                                        [[-9.42606,952.141,714.465],[0.876922,0.168711,0.443186,0.0782947],[-1,1,-1,1],[5409.45,9E+09,9E+09,9E+09,9E+09,9E+09]],
                                        [[-9.41231,953.154,714.855],[0.877775,0.167301,0.442197,0.0773528],[-1,1,-1,1],[5407.45,9E+09,9E+09,9E+09,9E+09,9E+09]],
                                        [[-9.39801,954.16,715.244],[0.878624,0.16588,0.441207,0.0764259],[-1,1,-1,1],[5405.45,9E+09,9E+09,9E+09,9E+09,9E+09]],
                                        [[-9.38345,955.166,715.628],[0.879465,0.16447,0.440214,0.0755183],[-1,1,-1,1],[5403.45,9E+09,9E+09,9E+09,9E+09,9E+09]],
                                        [[-9.3692,956.176,716.011],[0.8803,0.163055,0.43922,0.0746309],[-1,1,-1,1],[5401.45,9E+09,9E+09,9E+09,9E+09,9E+09]],
                                        [[-9.35551,957.184,716.389],[0.881131,0.161641,0.438224,0.0737555],[-1,1,-1,1],[5399.45,9E+09,9E+09,9E+09,9E+09,9E+09]],
                                        [[-9.34535,958.198,716.761],[0.881958,0.160216,0.437227,0.0728897],[-1,1,-1,1],[5397.45,9E+09,9E+09,9E+09,9E+09,9E+09]],
                                        [[-9.33447,959.205,717.131],[0.882781,0.158787,0.436228,0.0720344],[-1,1,-1,1],[5395.45,9E+09,9E+09,9E+09,9E+09,9E+09]],
                                        [[-9.32008,960.217,717.498],[0.883599,0.157353,0.435228,0.0711963],[-1,1,-1,1],[5393.45,9E+09,9E+09,9E+09,9E+09,9E+09]],
                                        [[-9.30747,961.231,717.863],[0.884416,0.155903,0.434226,0.070355],[-1,1,-1,1],[5391.45,9E+09,9E+09,9E+09,9E+09,9E+09]],
                                        [[-9.29394,962.246,718.223],[0.885229,0.154452,0.433221,0.0695209],[-1,1,-1,1],[5389.45,9E+09,9E+09,9E+09,9E+09,9E+09]],
                                        [[-9.27922,963.255,718.579],[0.88604,0.152992,0.432214,0.0686898],[-1,1,-1,1],[5387.45,9E+09,9E+09,9E+09,9E+09,9E+09]],
                                        [[-9.26511,964.273,718.932],[0.886848,0.151509,0.431207,0.0678638],[-1,1,-1,1],[5385.45,9E+09,9E+09,9E+09,9E+09,9E+09]],
                                        [[-9.25676,965.291,719.283],[0.887657,0.15,0.4302,0.0670376],[-1,1,-1,1],[5383.45,9E+09,9E+09,9E+09,9E+09,9E+09]],
                                        [[-9.24412,966.308,719.631],[0.888456,0.148507,0.429189,0.0662374],[-1,1,-1,1],[5381.45,9E+09,9E+09,9E+09,9E+09,9E+09]],
                                        [[-9.23401,967.325,719.976],[0.889257,0.146977,0.428179,0.0654321],[-1,1,-1,1],[5379.45,9E+09,9E+09,9E+09,9E+09,9E+09]],
                                        [[-9.22588,968.345,720.318],[0.890054,0.145446,0.427167,0.064639],[-1,1,-1,1],[5377.45,9E+09,9E+09,9E+09,9E+09,9E+09]],
                                        [[-9.21433,969.364,720.656],[0.890847,0.143908,0.426152,0.0638457],[-1,1,-1,1],[5375.45,9E+09,9E+09,9E+09,9E+09,9E+09]],
                                        [[-9.20663,970.383,720.989],[0.891638,0.142368,0.425133,0.0630512],[-1,1,-1,1],[5373.45,9E+09,9E+09,9E+09,9E+09,9E+09]],
                                        [[-9.19797,971.403,721.317],[0.892429,0.140797,0.424113,0.0622536],[-1,1,-1,1],[5371.45,9E+09,9E+09,9E+09,9E+09,9E+09]],
                                        [[-9.18923,972.429,721.644],[0.893216,0.139218,0.423091,0.061457],[-1,1,-1,1],[5369.45,9E+09,9E+09,9E+09,9E+09,9E+09]],
                                        [[-9.18339,973.457,721.968],[0.894004,0.13761,0.422068,0.0606508],[-1,1,-1,1],[5367.45,9E+09,9E+09,9E+09,9E+09,9E+09]],
                                        [[-9.1751,974.477,722.287],[0.894787,0.13601,0.42104,0.0598502],[-1,1,-1,1],[5365.45,9E+09,9E+09,9E+09,9E+09,9E+09]],
                                        [[-9.1676,975.509,722.603],[0.895569,0.134397,0.420009,0.0590409],[-1,1,-1,1],[5363.45,9E+09,9E+09,9E+09,9E+09,9E+09]],
                                        [[-9.15948,976.535,722.914],[0.896348,0.132767,0.418977,0.0582357],[-1,1,-1,1],[5361.45,9E+09,9E+09,9E+09,9E+09,9E+09]],
                                        [[-9.15505,977.568,723.219],[0.897127,0.131111,0.417943,0.0574251],[-1,1,-1,1],[5359.45,9E+09,9E+09,9E+09,9E+09,9E+09]],
                                        [[-9.1446,978.598,723.524],[0.897904,0.129432,0.416907,0.056606],[-1,1,-1,1],[5357.45,9E+09,9E+09,9E+09,9E+09,9E+09]],
                                        [[-9.1363,979.625,723.822],[0.898678,0.127747,0.415867,0.0557895],[-1,1,-1,1],[5355.45,9E+09,9E+09,9E+09,9E+09,9E+09]],
                                        [[-9.1268,980.66,724.115],[0.899451,0.126043,0.414825,0.0549606],[-1,1,-1,1],[5353.45,9E+09,9E+09,9E+09,9E+09,9E+09]],
                                        [[-9.12389,981.693,724.406],[0.900221,0.12434,0.413778,0.0541259],[-1,1,-1,1],[5351.45,9E+09,9E+09,9E+09,9E+09,9E+09]],
                                        [[-9.12032,982.72,724.689],[0.900987,0.12262,0.41273,0.0532925],[-1,1,-1,1],[5349.45,9E+09,9E+09,9E+09,9E+09,9E+09]],
                                        [[-9.11677,983.752,724.97],[0.90175,0.120895,0.411678,0.0524628],[-1,1,-1,1],[5347.45,9E+09,9E+09,9E+09,9E+09,9E+09]],
                                        [[-9.11474,984.782,725.248],[0.902507,0.119183,0.410621,0.0516391],[-1,1,-1,1],[5345.45,9E+09,9E+09,9E+09,9E+09,9E+09]],
                                        [[-9.11064,985.807,725.519],[0.903261,0.11746,0.409561,0.0508105],[-1,1,-1,1],[5343.45,9E+09,9E+09,9E+09,9E+09,9E+09]],
                                        [[-9.10221,986.836,725.788],[0.90401,0.115747,0.408497,0.0499893],[-1,1,-1,1],[5341.45,9E+09,9E+09,9E+09,9E+09,9E+09]],
                                        [[-9.09653,987.866,726.051],[0.904755,0.114033,0.407429,0.0491646],[-1,1,-1,1],[5339.45,9E+09,9E+09,9E+09,9E+09,9E+09]],
                                        [[-9.09416,988.889,726.31],[0.905493,0.112332,0.406357,0.0483544],[-1,1,-1,1],[5337.45,9E+09,9E+09,9E+09,9E+09,9E+09]],
                                        [[-9.09093,989.917,726.564],[0.90623,0.1106,0.405284,0.0475387],[-1,1,-1,1],[5335.45,9E+09,9E+09,9E+09,9E+09,9E+09]],
                                        [[-9.08773,990.947,726.814],[0.906959,0.108888,0.404207,0.0467441],[-1,1,-1,1],[5333.45,9E+09,9E+09,9E+09,9E+09,9E+09]],
                                        [[-9.08435,991.974,727.061],[0.907685,0.107163,0.403128,0.0459566],[-1,1,-1,1],[5331.45,9E+09,9E+09,9E+09,9E+09,9E+09]],
                                        [[-9.07911,993.002,727.303],[0.908405,0.105442,0.402046,0.0451818],[-1,1,-1,1],[5329.45,9E+09,9E+09,9E+09,9E+09,9E+09]],
                                        [[-9.07648,994.024,727.537],[0.909122,0.103706,0.400962,0.0444079],[-1,1,-1,1],[5327.45,9E+09,9E+09,9E+09,9E+09,9E+09]],
                                        [[-9.07295,995.05,727.768],[0.909833,0.101981,0.399873,0.0436403],[-1,1,-1,1],[5325.45,9E+09,9E+09,9E+09,9E+09,9E+09]],
                                        [[-9.07148,996.075,727.994],[0.910541,0.100239,0.398783,0.0428822],[-1,1,-1,1],[5323.45,9E+09,9E+09,9E+09,9E+09,9E+09]],
                                        [[-9.0704,997.101,728.218],[0.911243,0.0985139,0.397688,0.0421237],[-1,1,-1,1],[5321.45,9E+09,9E+09,9E+09,9E+09,9E+09]],
                                        [[-9.0673,998.127,728.437],[0.91194,0.0967962,0.39659,0.0413749],[-1,1,-1,1],[5319.45,9E+09,9E+09,9E+09,9E+09,9E+09]],
                                        [[-9.06497,999.147,728.652],[0.912634,0.0950637,0.395489,0.0406237],[-1,1,-1,1],[5317.45,9E+09,9E+09,9E+09,9E+09,9E+09]],
                                        [[-9.06877,1000.17,728.866],[0.913321,0.0933469,0.394385,0.0398957],[-1,1,-1,1],[5315.45,9E+09,9E+09,9E+09,9E+09,9E+09]],
                                        [[-9.06649,1001.2,729.076],[0.914004,0.0916219,0.393278,0.0391674],[-1,1,-1,1],[5313.45,9E+09,9E+09,9E+09,9E+09,9E+09]],
                                        [[-9.06642,1002.21,729.283],[0.914682,0.0899032,0.392168,0.0384524],[-1,1,-1,1],[5311.45,9E+09,9E+09,9E+09,9E+09,9E+09]],
                                        [[-9.06462,1003.24,729.485],[0.915354,0.0881878,0.391055,0.0377523],[-1,1,-1,1],[5309.45,9E+09,9E+09,9E+09,9E+09,9E+09]],
                                        [[-9.06208,1004.26,729.685],[0.916021,0.0864863,0.389938,0.0370562],[-1,1,-1,1],[5307.45,9E+09,9E+09,9E+09,9E+09,9E+09]],
                                        [[-9.0617,1005.28,729.877],[0.916684,0.0847922,0.388818,0.0363613],[-1,1,-1,1],[5305.45,9E+09,9E+09,9E+09,9E+09,9E+09]],
                                        [[-9.0618,1006.3,730.067],[0.917341,0.0831071,0.387694,0.0356762],[-1,1,-1,1],[5303.45,9E+09,9E+09,9E+09,9E+09,9E+09]],
                                        [[-9.06366,1007.33,730.253],[0.917994,0.0814151,0.386568,0.0349967],[-1,1,-1,1],[5301.45,9E+09,9E+09,9E+09,9E+09,9E+09]],
                                        [[-9.06773,1008.35,730.436],[0.918642,0.0797262,0.385438,0.0343187],[-1,1,-1,1],[5299.45,9E+09,9E+09,9E+09,9E+09,9E+09]],
                                        [[-9.06962,1009.38,730.613],[0.919287,0.078025,0.384306,0.0336379],[-1,1,-1,1],[5297.45,9E+09,9E+09,9E+09,9E+09,9E+09]],
                                        [[-9.07396,1010.41,730.785],[0.919927,0.0763415,0.38317,0.0329695],[-1,1,-1,1],[5295.45,9E+09,9E+09,9E+09,9E+09,9E+09]],
                                        [[-9.07654,1011.44,730.954],[0.920562,0.0746653,0.382031,0.0322975],[-1,1,-1,1],[5293.45,9E+09,9E+09,9E+09,9E+09,9E+09]],
                                        [[-9.07826,1012.47,731.121],[0.921193,0.0729844,0.380888,0.0316208],[-1,1,-1,1],[5291.45,9E+09,9E+09,9E+09,9E+09,9E+09]],
                                        [[-9.08255,1013.5,731.281],[0.92182,0.0713165,0.379742,0.0309445],[-1,1,-1,1],[5289.45,9E+09,9E+09,9E+09,9E+09,9E+09]],
                                        [[-9.08421,1014.53,731.44],[0.922442,0.0696605,0.378593,0.030272],[-1,1,-1,1],[5287.45,9E+09,9E+09,9E+09,9E+09,9E+09]],
                                        [[-9.08975,1015.56,731.596],[0.923059,0.0680076,0.37744,0.0295963],[-1,1,-1,1],[5285.45,9E+09,9E+09,9E+09,9E+09,9E+09]],
                                        [[-9.0966,1016.6,731.748],[0.923671,0.0663727,0.376284,0.0289251],[-1,1,-1,1],[5283.45,9E+09,9E+09,9E+09,9E+09,9E+09]],
                                        [[-9.10215,1017.64,731.899],[0.924279,0.0647426,0.375124,0.0282482],[-1,1,-1,1],[5281.45,9E+09,9E+09,9E+09,9E+09,9E+09]],
                                        [[-9.10383,1018.68,732.045],[0.924768,0.0630968,0.374247,0.0276039],[-1,1,-1,1],[5279.45,9E+09,9E+09,9E+09,9E+09,9E+09]],
                                        [[-9.10862,1019.71,732.189],[0.925235,0.0614779,0.373407,0.0269648],[-1,1,-1,1],[5277.45,9E+09,9E+09,9E+09,9E+09,9E+09]],
                                        [[-9.11369,1020.75,732.329],[0.925702,0.0598716,0.372556,0.0263164],[-1,1,-1,1],[5275.45,9E+09,9E+09,9E+09,9E+09,9E+09]],
                                        [[-9.11508,1021.79,732.464],[0.926177,0.0583058,0.37167,0.0256666],[-1,1,-1,1],[5273.45,9E+09,9E+09,9E+09,9E+09,9E+09]],
                                        [[-9.1214,1022.83,732.596],[0.926762,0.0567618,0.370495,0.0249872],[-1,1,-1,1],[5271.45,9E+09,9E+09,9E+09,9E+09,9E+09]],
                                        [[-9.12894,1023.88,732.723],[0.927343,0.0552133,0.369318,0.0243044],[-1,1,-1,1],[5269.45,9E+09,9E+09,9E+09,9E+09,9E+09]],
                                        [[-9.13472,1024.93,732.844],[0.92792,0.0536729,0.368138,0.0236249],[-1,1,-1,1],[5267.45,9E+09,9E+09,9E+09,9E+09,9E+09]],
                                        [[-9.13867,1025.98,732.963],[0.928493,0.0521304,0.366956,0.0229502],[-1,1,-1,1],[5265.45,9E+09,9E+09,9E+09,9E+09,9E+09]],
                                        [[-9.14382,1027.04,733.081],[0.929061,0.050589,0.365772,0.0222821],[-1,1,-1,1],[5263.45,9E+09,9E+09,9E+09,9E+09,9E+09]],
                                        [[-9.1507,1028.08,733.194],[0.929626,0.0490426,0.364587,0.0216121],[-1,1,-1,1],[5261.45,9E+09,9E+09,9E+09,9E+09,9E+09]],
                                        [[-9.15559,1029.14,733.305],[0.930187,0.0474902,0.363399,0.0209453],[-1,1,-1,1],[5259.45,9E+09,9E+09,9E+09,9E+09,9E+09]],
                                        [[-9.15988,1030.2,733.412],[0.930743,0.0459461,0.362209,0.02029],[-1,1,-1,1],[5257.45,9E+09,9E+09,9E+09,9E+09,9E+09]],
                                        [[-9.16456,1031.25,733.519],[0.931295,0.0443892,0.361018,0.0196283],[-1,1,-1,1],[5255.45,9E+09,9E+09,9E+09,9E+09,9E+09]],
                                        [[-9.16908,1032.31,733.624],[0.931732,0.0428385,0.36011,0.0189873],[-1,1,-1,1],[5253.45,9E+09,9E+09,9E+09,9E+09,9E+09]],
                                        [[-9.17239,1033.37,733.724],[0.932041,0.0412613,0.359528,0.0183526],[-1,1,-1,1],[5251.45,9E+09,9E+09,9E+09,9E+09,9E+09]],
                                        [[-9.17859,1034.43,733.818],[0.932224,0.0396543,0.359265,0.0177331],[-1,1,-1,1],[5249.45,9E+09,9E+09,9E+09,9E+09,9E+09]],
                                        [[-9.18245,1035.49,733.91],[0.932293,0.0380624,0.359288,0.0171463],[-1,1,-1,1],[5247.45,9E+09,9E+09,9E+09,9E+09,9E+09]],
                                        [[-9.19017,1036.55,733.998],[0.93236,0.0364388,0.359311,0.016547],[-1,1,-1,1],[5245.45,9E+09,9E+09,9E+09,9E+09,9E+09]],
                                        [[-9.19466,1037.61,734.082],[0.932424,0.0348098,0.359332,0.0159428],[-1,1,-1,1],[5243.45,9E+09,9E+09,9E+09,9E+09,9E+09]],
                                        [[-9.1953,1038.67,734.166],[0.932486,0.0331789,0.359352,0.0153449],[-1,1,-1,1],[5241.45,9E+09,9E+09,9E+09,9E+09,9E+09]],
                                        [[-9.19697,1039.73,734.244],[0.932545,0.0315386,0.359372,0.0147493],[-1,1,-1,1],[5239.45,9E+09,9E+09,9E+09,9E+09,9E+09]],
                                        [[-9.19883,1040.79,734.318],[0.9326,0.0299119,0.35939,0.0141594],[-1,1,-1,1],[5237.45,9E+09,9E+09,9E+09,9E+09,9E+09]],
                                        [[-9.20468,1041.85,734.386],[0.932654,0.0282568,0.359407,0.0135601],[-1,1,-1,1],[5235.45,9E+09,9E+09,9E+09,9E+09,9E+09]],
                                        [[-9.21101,1042.92,734.45],[0.932705,0.0266084,0.359424,0.0129718],[-1,1,-1,1],[5233.45,9E+09,9E+09,9E+09,9E+09,9E+09]],
                                        [[-9.21839,1043.99,734.512],[0.932753,0.0249497,0.359439,0.012381],[-1,1,-1,1],[5231.45,9E+09,9E+09,9E+09,9E+09,9E+09]],
                                        [[-9.22355,1045.05,734.568],[0.932799,0.0232681,0.359453,0.0117858],[-1,1,-1,1],[5229.45,9E+09,9E+09,9E+09,9E+09,9E+09]],
                                        [[-9.2288,1046.11,734.619],[0.932842,0.0215742,0.359465,0.0111768],[-1,1,-1,1],[5227.45,9E+09,9E+09,9E+09,9E+09,9E+09]],
                                        [[-9.23402,1047.18,734.67],[0.932882,0.0198826,0.359477,0.0105783],[-1,1,-1,1],[5225.45,9E+09,9E+09,9E+09,9E+09,9E+09]],
                                        [[-9.24194,1048.24,734.717],[0.93292,0.0181553,0.359487,0.00997164],[-1,1,-1,1],[5223.45,9E+09,9E+09,9E+09,9E+09,9E+09]],
                                        [[-9.24738,1049.3,734.759],[0.932955,0.0164235,0.359497,0.0093672],[-1,1,-1,1],[5221.45,9E+09,9E+09,9E+09,9E+09,9E+09]],
                                        [[-9.25195,1050.36,734.796],[0.932986,0.0147083,0.359504,0.00876838],[-1,1,-1,1],[5219.45,9E+09,9E+09,9E+09,9E+09,9E+09]],
                                        [[-9.25835,1051.43,734.832],[0.933015,0.0129844,0.359511,0.00817269],[-1,1,-1,1],[5217.45,9E+09,9E+09,9E+09,9E+09,9E+09]],
                                        [[-9.26627,1052.49,734.862],[0.93304,0.0112621,0.359515,0.00757162],[-1,1,-1,1],[5215.45,9E+09,9E+09,9E+09,9E+09,9E+09]],
                                        [[-9.27436,1053.55,734.885],[0.933063,0.00953464,0.359519,0.00697427],[-1,1,-1,1],[5213.45,9E+09,9E+09,9E+09,9E+09,9E+09]],
                                        [[-9.27864,1054.61,734.905],[0.933082,0.00781355,0.359521,0.0063799],[-1,1,-1,1],[5211.45,9E+09,9E+09,9E+09,9E+09,9E+09]],
                                        [[-9.28602,1055.67,734.922],[0.933099,0.00607636,0.359522,0.00578946],[-1,1,-1,1],[5209.45,9E+09,9E+09,9E+09,9E+09,9E+09]],
                                        [[-9.29461,1056.73,734.934],[0.933112,0.00434153,0.359521,0.00520004],[-1,1,-1,1],[5207.45,9E+09,9E+09,9E+09,9E+09,9E+09]],
                                        [[-9.30256,1057.79,734.945],[0.933123,0.0026124,0.359519,0.00459857],[-1,1,-1,1],[5205.45,9E+09,9E+09,9E+09,9E+09,9E+09]],
                                        [[-9.31218,1058.84,734.953],[0.93313,0.000907263,0.359516,0.00399223],[-1,1,-1,1],[5203.45,9E+09,9E+09,9E+09,9E+09,9E+09]],
                                        [[-9.31758,1059.9,734.959],[0.933135,-0.000803467,0.359511,0.0033728],[-1,1,-1,1],[5201.45,9E+09,9E+09,9E+09,9E+09,9E+09]],
                                        [[-9.32476,1060.95,734.959],[0.933136,-0.00252175,0.359504,0.00274454],[-1,1,-1,1],[5199.45,9E+09,9E+09,9E+09,9E+09,9E+09]],
                                        [[-9.33054,1062.01,734.952],[0.933134,-0.00424319,0.359497,0.00211743],[-1,1,-1,1],[5197.45,9E+09,9E+09,9E+09,9E+09,9E+09]],
                                        [[-9.33972,1063.06,734.944],[0.93313,-0.00595179,0.359488,0.00149342],[-1,1,-1,1],[5195.45,9E+09,9E+09,9E+09,9E+09,9E+09]],
                                        [[-9.34233,1064.11,734.933],[0.933122,-0.00769029,0.359478,0.000857251],[-1,1,-1,1],[5193.45,9E+09,9E+09,9E+09,9E+09,9E+09]],
                                        [[-9.35049,1065.16,734.916],[0.933111,-0.00941787,0.359466,0.000226595],[-1,1,-1,1],[5191.45,9E+09,9E+09,9E+09,9E+09,9E+09]],
                                        [[-9.35937,1066.21,734.892],[0.933096,-0.0111453,0.359453,-0.000399761],[-1,1,-1,1],[5189.45,9E+09,9E+09,9E+09,9E+09,9E+09]],
                                        [[-9.36839,1067.26,734.868],[0.933079,-0.0128686,0.359439,-0.00101946],[-1,1,-1,1],[5187.45,9E+09,9E+09,9E+09,9E+09,9E+09]],
                                        [[-9.3753,1068.31,734.843],[0.933059,-0.0145855,0.359423,-0.00163268],[-1,1,-1,1],[5185.45,9E+09,9E+09,9E+09,9E+09,9E+09]],
                                        [[-9.38546,1069.36,734.811],[0.933036,-0.0163006,0.359407,-0.00226047],[-1,1,-1,1],[5183.45,9E+09,9E+09,9E+09,9E+09,9E+09]],
                                        [[-9.3921,1070.4,734.774],[0.93301,-0.0179895,0.359389,-0.00288911],[-1,1,-1,1],[5181.45,9E+09,9E+09,9E+09,9E+09,9E+09]],
                                        [[-9.40082,1071.45,734.737],[0.932981,-0.0196682,0.35937,-0.00351875],[-1,1,-1,1],[5179.45,9E+09,9E+09,9E+09,9E+09,9E+09]],
                                        [[-9.4099,1072.49,734.694],[0.932949,-0.0213521,0.35935,-0.00414987],[-1,1,-1,1],[5177.45,9E+09,9E+09,9E+09,9E+09,9E+09]],
                                        [[-9.41928,1073.54,734.646],[0.932914,-0.0230319,0.359329,-0.00480232],[-1,1,-1,1],[5175.45,9E+09,9E+09,9E+09,9E+09,9E+09]],
                                        [[-9.42784,1074.58,734.594],[0.932876,-0.0246908,0.359308,-0.0054537],[-1,1,-1,1],[5173.45,9E+09,9E+09,9E+09,9E+09,9E+09]],
                                        [[-9.43497,1075.63,734.54],[0.932835,-0.0263633,0.359285,-0.00611693],[-1,1,-1,1],[5171.45,9E+09,9E+09,9E+09,9E+09,9E+09]],
                                        [[-9.44138,1076.67,734.485],[0.932792,-0.0280014,0.359262,-0.00677309],[-1,1,-1,1],[6236.68,9E+09,9E+09,9E+09,9E+09,9E+09]],
                                        [[-9.44917,1077.72,734.421],[0.932746,-0.0296326,0.359238,-0.00743051],[-1,1,-1,1],[6236.68,9E+09,9E+09,9E+09,9E+09,9E+09]],
                                        [[-9.45523,1078.76,734.355],[0.932697,-0.0312312,0.359214,-0.00809553],[-1,1,-1,1],[6236.68,9E+09,9E+09,9E+09,9E+09,9E+09]],
                                        [[-9.46422,1079.81,734.283],[0.932647,-0.0328114,0.35919,-0.00875125],[-1,1,-1,1],[6236.68,9E+09,9E+09,9E+09,9E+09,9E+09]],
                                        [[-9.47057,1080.85,734.209],[0.932593,-0.0344018,0.359164,-0.00941589],[-1,1,-1,1],[6236.68,9E+09,9E+09,9E+09,9E+09,9E+09]],
                                        [[-9.47968,1081.89,734.129],[0.932536,-0.0359863,0.359138,-0.0100824],[-1,1,-1,1],[6236.68,9E+09,9E+09,9E+09,9E+09,9E+09]],
                                        [[-9.4897,1082.94,734.047],[0.932477,-0.0375478,0.359111,-0.0107548],[-1,1,-1,1],[6236.68,9E+09,9E+09,9E+09,9E+09,9E+09]],
                                        [[-9.5013,1083.98,733.964],[0.932416,-0.0390866,0.359085,-0.0114251],[-1,1,-1,1],[6236.68,9E+09,9E+09,9E+09,9E+09,9E+09]],
                                        [[-9.51069,1085.02,733.876],[0.932352,-0.0406395,0.359057,-0.0121043],[-1,1,-1,1],[6236.68,9E+09,9E+09,9E+09,9E+09,9E+09]],
                                        [[-9.52236,1086.06,733.783],[0.932285,-0.0421839,0.359029,-0.0127787],[-1,1,-1,1],[6236.68,9E+09,9E+09,9E+09,9E+09,9E+09]],
                                        [[-9.52751,1087.11,733.689],[0.932216,-0.0437178,0.359,-0.0134556],[-1,1,-1,1],[6236.68,9E+09,9E+09,9E+09,9E+09,9E+09]],
                                        [[-9.53247,1088.15,733.595],[0.932144,-0.0452455,0.358971,-0.0141268],[-1,1,-1,1],[6236.68,9E+09,9E+09,9E+09,9E+09,9E+09]],
                                        [[-9.53836,1089.2,733.494],[0.93207,-0.0467678,0.358941,-0.014803],[-1,1,-1,1],[6236.68,9E+09,9E+09,9E+09,9E+09,9E+09]],
                                        [[-9.54597,1090.24,733.388],[0.985491,-0.093353,0.141246,-0.0119022],[-1,1,-1,1],[6236.68,9E+09,9E+09,9E+09,9E+09,9E+09]],
                                        [[-9.54803,1091.29,733.28],[0.985491,-0.093353,0.141246,-0.0119022],[-1,1,-1,1],[6236.68,9E+09,9E+09,9E+09,9E+09,9E+09]],
                                        [[-9.55346,1092.33,733.169],[0.985491,-0.093353,0.141246,-0.0119022],[-1,1,-1,1],[6236.68,9E+09,9E+09,9E+09,9E+09,9E+09]],
                                        [[-9.55735,1093.38,733.054],[0.985491,-0.093353,0.141246,-0.0119022],[-1,2,-1,1],[6236.68,9E+09,9E+09,9E+09,9E+09,9E+09]],
                                        [[-9.56203,1094.43,732.939],[0.985491,-0.093353,0.141246,-0.0119022],[-1,2,-1,1],[6236.68,9E+09,9E+09,9E+09,9E+09,9E+09]],
                                        [[-9.5657,1095.48,732.819],[0.985491,-0.093353,0.141246,-0.0119022],[-1,2,-1,1],[6236.68,9E+09,9E+09,9E+09,9E+09,9E+09]],
                                        [[-9.56666,1096.53,732.694],[0.985491,-0.093353,0.141246,-0.0119022],[-1,2,-1,1],[6236.68,9E+09,9E+09,9E+09,9E+09,9E+09]],
                                        [[-9.57459,1097.59,732.566],[0.985491,-0.093353,0.141246,-0.0119022],[-1,2,-1,1],[6236.68,9E+09,9E+09,9E+09,9E+09,9E+09]],
                                        [[-9.5814,1098.64,732.433],[0.985491,-0.093353,0.141246,-0.0119022],[-1,2,-1,1],[6236.68,9E+09,9E+09,9E+09,9E+09,9E+09]],
                                        [[-9.58484,1099.7,732.296],[0.985491,-0.093353,0.141246,-0.0119022],[-1,2,-1,1],[6236.68,9E+09,9E+09,9E+09,9E+09,9E+09]],
                                        [[-9.59047,1100.75,732.156],[0.985491,-0.093353,0.141246,-0.0119022],[-1,2,-1,1],[6236.68,9E+09,9E+09,9E+09,9E+09,9E+09]],
                                        [[-9.59372,1101.8,732.01],[0.985491,-0.093353,0.141246,-0.0119022],[-1,2,-1,1],[6236.68,9E+09,9E+09,9E+09,9E+09,9E+09]],
                                        [[-9.59735,1102.85,731.863],[0.985491,-0.093353,0.141246,-0.0119022],[-1,2,-1,1],[6236.68,9E+09,9E+09,9E+09,9E+09,9E+09]],
                                        [[-9.60241,1103.9,731.714],[0.985491,-0.093353,0.141246,-0.0119022],[-1,2,-1,1],[6236.68,9E+09,9E+09,9E+09,9E+09,9E+09]],
                                        [[-9.60621,1104.95,731.557],[0.985491,-0.093353,0.141246,-0.0119022],[-1,2,-1,1],[6236.68,9E+09,9E+09,9E+09,9E+09,9E+09]],
                                        [[-9.61035,1106,731.399],[0.985491,-0.093353,0.141246,-0.0119022],[-1,2,-1,1],[6236.68,9E+09,9E+09,9E+09,9E+09,9E+09]],
                                        [[-9.61369,1107.04,731.237],[0.985491,-0.093353,0.141246,-0.0119022],[-1,2,-1,1],[6236.68,9E+09,9E+09,9E+09,9E+09,9E+09]],
                                        [[-9.58778,1107.96,731.564],[0.985491,-0.093353,0.141246,-0.0119022],[-1,2,-1,1],[6236.68,9E+09,9E+09,9E+09,9E+09,9E+09]],
                                        [[-9.63993,1108.93,731.47],[0.985491,-0.093353,0.141246,-0.0119022],[-1,2,-1,1],[6236.68,9E+09,9E+09,9E+09,9E+09,9E+09]],
                                        [[-9.67296,1110.16,731.223],[0.985491,-0.093353,0.141246,-0.0119022],[-1,2,-1,1],[6236.68,9E+09,9E+09,9E+09,9E+09,9E+09]],
                                        [[-9.71324,1111.24,731.006],[0.985491,-0.093353,0.141246,-0.0119022],[-1,2,-1,1],[6236.68,9E+09,9E+09,9E+09,9E+09,9E+09]],
                                        [[-9.55261,1112.24,730.878],[0.985491,-0.093353,0.141246,-0.0119022],[-1,2,-1,1],[6236.68,9E+09,9E+09,9E+09,9E+09,9E+09]],
                                        [[-9.59298,1113.23,730.702],[0.985491,-0.093353,0.141246,-0.0119022],[-1,2,-1,1],[6236.68,9E+09,9E+09,9E+09,9E+09,9E+09]],
                                        [[-9.60242,1114.22,730.493],[0.985491,-0.093353,0.141246,-0.0119022],[-1,2,-1,1],[6236.68,9E+09,9E+09,9E+09,9E+09,9E+09]],
                                        [[-9.67186,1115.48,730.435],[0.985491,-0.093353,0.141246,-0.0119022],[-1,2,-1,1],[6236.68,9E+09,9E+09,9E+09,9E+09,9E+09]],
                                        [[-9.60473,1116.61,730.195],[0.985491,-0.093353,0.141246,-0.0119022],[-1,2,-1,1],[6236.68,9E+09,9E+09,9E+09,9E+09,9E+09]],
                                        [[-9.57755,1117.77,729.904],[0.985491,-0.093353,0.141246,-0.0119022],[-1,2,-1,1],[6236.68,9E+09,9E+09,9E+09,9E+09,9E+09]],
                                        [[-9.7523,1118.85,729.748],[0.985491,-0.093353,0.141246,-0.0119022],[-1,2,-1,1],[6236.68,9E+09,9E+09,9E+09,9E+09,9E+09]],
                                        [[-9.66734,1119.87,729.548],[0.985491,-0.093353,0.141246,-0.0119022],[-1,2,-1,1],[6236.68,9E+09,9E+09,9E+09,9E+09,9E+09]],
                                        [[-9.61121,1121.05,729.204],[0.985491,-0.093353,0.141246,-0.0119022],[-1,2,-1,1],[6236.68,9E+09,9E+09,9E+09,9E+09,9E+09]],
                                        [[-9.70925,1121.92,729.016],[0.985491,-0.093353,0.141246,-0.0119022],[-1,2,-1,1],[6236.68,9E+09,9E+09,9E+09,9E+09,9E+09]],
                                        [[-9.66673,1122.8,728.731],[0.985491,-0.093353,0.141246,-0.0119022],[-1,2,-1,1],[6236.68,9E+09,9E+09,9E+09,9E+09,9E+09]],
                                        [[-9.69603,1123.7,728.667],[0.985491,-0.093353,0.141246,-0.0119022],[-1,2,-1,1],[6236.68,9E+09,9E+09,9E+09,9E+09,9E+09]],
                                        [[-9.75339,1124.68,728.438],[0.985491,-0.093353,0.141246,-0.0119022],[-1,2,-1,1],[6236.68,9E+09,9E+09,9E+09,9E+09,9E+09]],
                                        [[-9.71084,1125.94,728.144],[0.985491,-0.093353,0.141246,-0.0119022],[-1,2,-1,1],[6236.68,9E+09,9E+09,9E+09,9E+09,9E+09]],
                                        [[-9.73429,1126.89,727.945],[0.985491,-0.093353,0.141246,-0.0119022],[-1,2,-1,1],[6236.68,9E+09,9E+09,9E+09,9E+09,9E+09]],
                                        [[-9.6781,1127.86,727.8],[0.985491,-0.093353,0.141246,-0.0119022],[-1,2,-1,1],[6236.68,9E+09,9E+09,9E+09,9E+09,9E+09]],
                                        [[-7.75832,1127.97,730.662],[0.992368,-0.0953153,0.0782395,-0.000133741],[-1,2,-1,1],[6236.68,9E+09,9E+09,9E+09,9E+09,9E+09]],
                                        [[-7.81515,1128.99,730.391],[0.992368,-0.0953153,0.0782395,-0.000133741],[-1,2,-1,1],[6236.68,9E+09,9E+09,9E+09,9E+09,9E+09]],
                                        [[-7.76771,1129.99,730.16],[0.992368,-0.0953153,0.0782395,-0.000133741],[-1,2,-1,1],[6236.68,9E+09,9E+09,9E+09,9E+09,9E+09]],
                                        [[-7.81261,1130.96,729.847],[0.992368,-0.0953153,0.0782395,-0.000133741],[-1,2,-1,1],[6236.68,9E+09,9E+09,9E+09,9E+09,9E+09]],
                                        [[-7.78007,1132.14,729.608],[0.992368,-0.0953153,0.0782395,-0.000133741],[-1,2,-1,1],[6236.68,9E+09,9E+09,9E+09,9E+09,9E+09]],
                                        [[-7.80198,1133.12,729.485],[0.992368,-0.0953153,0.0782395,-0.000133741],[-1,2,-1,1],[6236.68,9E+09,9E+09,9E+09,9E+09,9E+09]],
                                        [[-7.74667,1134.11,729.334],[0.992368,-0.0953153,0.0782395,-0.000133741],[-1,2,-1,1],[6236.68,9E+09,9E+09,9E+09,9E+09,9E+09]],
                                        [[-7.87265,1135.1,729.104],[0.992368,-0.0953153,0.0782395,-0.000133741],[-1,2,-1,1],[6236.68,9E+09,9E+09,9E+09,9E+09,9E+09]],
                                        [[-7.84835,1136.09,728.857],[0.992368,-0.0953153,0.0782395,-0.000133741],[-1,2,-1,1],[6236.68,9E+09,9E+09,9E+09,9E+09,9E+09]],
                                        [[-7.77784,1137.09,728.602],[0.992368,-0.0953153,0.0782395,-0.000133741],[-1,2,-1,1],[6236.68,9E+09,9E+09,9E+09,9E+09,9E+09]],
                                        [[-7.77233,1138.32,728.411],[0.992368,-0.0953153,0.0782395,-0.000133741],[-1,2,-1,1],[6236.68,9E+09,9E+09,9E+09,9E+09,9E+09]],
                                        [[-942.032,325.34,457.38],[0.703525,-0.0244225,-0.0246412,0.709823],[-1,0,-1,0],[0,9E+09,9E+09,9E+09,9E+09,9E+09]],
                                        [[-942.931,325.333,457.327],[0.703391,-0.0241448,-0.0243708,0.709974],[-1,0,-1,0],[0,9E+09,9E+09,9E+09,9E+09,9E+09]],
                                        [[-943.836,325.327,457.255],[0.703219,-0.0237819,-0.024017,0.710169],[-1,0,-1,0],[0,9E+09,9E+09,9E+09,9E+09,9E+09]],
                                        [[-944.756,325.317,457.198],[0.702977,-0.0234767,-0.0237256,0.710429],[-1,0,-1,0],[0,9E+09,9E+09,9E+09,9E+09,9E+09]],
                                        [[-945.675,325.302,457.136],[0.702567,-0.0232584,-0.0235325,0.710848],[-1,0,-1,0],[0,9E+09,9E+09,9E+09,9E+09,9E+09]],
                                        [[-946.582,325.293,457.084],[0.70177,-0.0231129,-0.0234381,0.711643],[-1,0,-1,0],[0,9E+09,9E+09,9E+09,9E+09,9E+09]],
                                        [[-947.482,325.283,457.032],[0.700367,-0.0228949,-0.023309,0.713035],[-1,0,-1,0],[0,9E+09,9E+09,9E+09,9E+09,9E+09]],
                                        [[-948.369,325.274,456.975],[0.698391,-0.0226104,-0.0231475,0.714984],[-1,0,-1,0],[0,9E+09,9E+09,9E+09,9E+09,9E+09]],
                                        [[-949.255,325.261,456.929],[0.694788,-0.0222582,-0.0230179,0.718501],[-1,0,-1,0],[0,9E+09,9E+09,9E+09,9E+09,9E+09]],
                                        [[-950.141,325.245,456.872],[0.689571,-0.021829,-0.0229039,0.723527],[-1,0,-1,0],[0,9E+09,9E+09,9E+09,9E+09,9E+09]],
                                        [[-951.049,325.226,456.819],[0.68273,-0.0213162,-0.0227922,0.730004],[-1,0,-1,0],[0,9E+09,9E+09,9E+09,9E+09,9E+09]],
                                        [[-951.944,325.211,456.76],[0.674269,-0.0207658,-0.0227237,0.737844],[-1,0,-1,0],[0,9E+09,9E+09,9E+09,9E+09,9E+09]],
                                        [[-952.862,325.189,456.7],[0.664178,-0.0201186,-0.0226262,0.746961],[-1,0,-1,0],[0,9E+09,9E+09,9E+09,9E+09,9E+09]],
                                        [[-953.741,325.166,456.655],[0.652502,-0.0194224,-0.022539,0.757203],[-1,0,-1,0],[0,9E+09,9E+09,9E+09,9E+09,9E+09]],
                                        [[-954.624,325.144,456.6],[1,0,0,0],[-1,0,-1,0],[0,9E+09,9E+09,9E+09,9E+09,9E+09]],
                                        [[-955.504,325.124,456.557],[1,0,0,0],[-1,0,-1,0],[0,9E+09,9E+09,9E+09,9E+09,9E+09]],
                                        [[-956.396,325.101,456.496],[1,0,0,0],[-1,0,-1,0],[0,9E+09,9E+09,9E+09,9E+09,9E+09]],
                                        [[-957.312,325.078,456.442],[1,0,0,0],[-1,0,-1,0],[0,9E+09,9E+09,9E+09,9E+09,9E+09]],
                                        [[-958.228,325.048,456.37],[1,0,0,0],[-1,0,-1,0],[0,9E+09,9E+09,9E+09,9E+09,9E+09]],
                                        [[-959.148,325.006,456.3],[1,0,0,0],[-1,0,-1,0],[0,9E+09,9E+09,9E+09,9E+09,9E+09]],
                                        [[-960.066,324.847,456.235],[1,0,0,0],[-1,0,-1,0],[0,9E+09,9E+09,9E+09,9E+09,9E+09]],
                                        [[-960.946,324.559,456.189],[1,0,0,0],[-1,0,-1,0],[0,9E+09,9E+09,9E+09,9E+09,9E+09]],
                                        [[-961.837,324.264,456.146],[1,0,0,0],[-1,0,-1,0],[0,9E+09,9E+09,9E+09,9E+09,9E+09]],
                                        [[-962.707,323.51,456.101],[1,0,0,0],[-1,0,-1,0],[0,9E+09,9E+09,9E+09,9E+09,9E+09]],
                                        [[-963.599,322.72,456.062],[1,0,0,0],[-1,0,-1,0],[0,9E+09,9E+09,9E+09,9E+09,9E+09]],
                                        [[-964.493,321.891,456.026],[1,0,0,0],[-1,0,-1,0],[0,9E+09,9E+09,9E+09,9E+09,9E+09]],
                                        [[-965.374,321.023,455.985],[1,0,0,0],[-1,0,-1,0],[0,9E+09,9E+09,9E+09,9E+09,9E+09]],
                                        [[-966.242,320.114,455.956],[1,0,0,0],[-1,0,-1,0],[0,9E+09,9E+09,9E+09,9E+09,9E+09]],
                                        [[-967.093,319.163,455.928],[1,0,0,0],[-1,0,-1,0],[0,9E+09,9E+09,9E+09,9E+09,9E+09]],
                                        [[-968.366,324.444,455.53],[1,0,0,0],[-1,0,-1,0],[0,9E+09,9E+09,9E+09,9E+09,9E+09]],
                                        [[-969.045,321.93,455.62],[1,0,0,0],[-1,0,-1,0],[0,9E+09,9E+09,9E+09,9E+09,9E+09]],
                                        [[-969.737,319.351,455.9],[1,0,0,0],[-1,0,-1,0],[0,9E+09,9E+09,9E+09,9E+09,9E+09]],
                                        [[-970.736,319.468,455.83],[1,0,0,0],[-1,0,-1,0],[0,9E+09,9E+09,9E+09,9E+09,9E+09]],
                                        [[-971.333,310.032,455.805],[1,0,0,0],[-1,0,-1,0],[0,9E+09,9E+09,9E+09,9E+09,9E+09]],
                                        [[-972.096,309.972,455.815],[1,0,0,0],[-1,0,-1,0],[0,9E+09,9E+09,9E+09,9E+09,9E+09]],
                                        [[-973.299,309.91,455.805],[1,0,0,0],[-1,0,-1,0],[0,9E+09,9E+09,9E+09,9E+09,9E+09]],
                                        [[-974.022,309.882,455.795],[1,0,0,0],[-1,0,-1,0],[0,9E+09,9E+09,9E+09,9E+09,9E+09]],
                                        [[-974.791,309.864,455.778],[1,0,0,0],[-1,0,-1,0],[0,9E+09,9E+09,9E+09,9E+09,9E+09]],
                                        [[-975.548,309.854,455.766],[1,0,0,0],[-1,0,-1,0],[0,9E+09,9E+09,9E+09,9E+09,9E+09]],
                                        [[0,0,0],[1,0,0,0],[0,-2,1,0],[0,9E+09,9E+09,9E+09,9E+09,9E+09]],
                                        [[0,0,0],[1,0,0,0],[0,-2,1,0],[0,9E+09,9E+09,9E+09,9E+09,9E+09]],
                                        [[0,0,0],[1,0,0,0],[0,-2,1,0],[0,9E+09,9E+09,9E+09,9E+09,9E+09]],
                                        [[0,0,0],[1,0,0,0],[0,-2,1,0],[0,9E+09,9E+09,9E+09,9E+09,9E+09]],
                                        [[0,0,0],[1,0,0,0],[0,-2,1,0],[0,9E+09,9E+09,9E+09,9E+09,9E+09]],
                                        [[0,0,0],[1,0,0,0],[0,-2,1,0],[0,9E+09,9E+09,9E+09,9E+09,9E+09]],
                                        [[0,0,0],[1,0,0,0],[0,-2,1,0],[0,9E+09,9E+09,9E+09,9E+09,9E+09]],
                                        [[0,0,0],[1,0,0,0],[0,-2,1,0],[0,9E+09,9E+09,9E+09,9E+09,9E+09]],
                                        [[0,0,0],[1,0,0,0],[0,-2,1,0],[0,9E+09,9E+09,9E+09,9E+09,9E+09]],
                                        [[0,0,0],[1,0,0,0],[0,-2,1,0],[0,9E+09,9E+09,9E+09,9E+09,9E+09]],
                                        [[0,0,0],[1,0,0,0],[0,-2,1,0],[0,9E+09,9E+09,9E+09,9E+09,9E+09]],
                                        [[0,0,0],[1,0,0,0],[0,-2,1,0],[0,9E+09,9E+09,9E+09,9E+09,9E+09]],
                                        [[0,0,0],[1,0,0,0],[0,-2,1,0],[0,9E+09,9E+09,9E+09,9E+09,9E+09]],
                                        [[0,0,0],[1,0,0,0],[0,-2,1,0],[0,9E+09,9E+09,9E+09,9E+09,9E+09]],
                                        [[0,0,0],[1,0,0,0],[0,-2,1,0],[0,9E+09,9E+09,9E+09,9E+09,9E+09]],
                                        [[0,0,0],[1,0,0,0],[0,-2,1,0],[0,9E+09,9E+09,9E+09,9E+09,9E+09]],
                                        [[0,0,0],[1,0,0,0],[0,-2,1,0],[0,9E+09,9E+09,9E+09,9E+09,9E+09]],
                                        [[0,0,0],[1,0,0,0],[0,-2,1,0],[0,9E+09,9E+09,9E+09,9E+09,9E+09]],
                                        [[0,0,0],[1,0,0,0],[0,-2,1,0],[0,9E+09,9E+09,9E+09,9E+09,9E+09]],
                                        [[0,0,0],[1,0,0,0],[0,-2,1,0],[0,9E+09,9E+09,9E+09,9E+09,9E+09]],
                                        [[0,0,0],[1,0,0,0],[0,-2,1,0],[0,9E+09,9E+09,9E+09,9E+09,9E+09]],
                                        [[0,0,0],[1,0,0,0],[0,-2,1,0],[0,9E+09,9E+09,9E+09,9E+09,9E+09]],
                                        [[0,0,0],[1,0,0,0],[0,-2,1,0],[0,9E+09,9E+09,9E+09,9E+09,9E+09]],
                                        [[0,0,0],[1,0,0,0],[0,-2,1,0],[0,9E+09,9E+09,9E+09,9E+09,9E+09]],
                                        [[0,0,0],[1,0,0,0],[0,-2,1,0],[0,9E+09,9E+09,9E+09,9E+09,9E+09]],
                                        [[0,0,0],[1,0,0,0],[0,-2,1,0],[0,9E+09,9E+09,9E+09,9E+09,9E+09]],
                                        [[0,0,0],[1,0,0,0],[0,-2,1,0],[0,9E+09,9E+09,9E+09,9E+09,9E+09]],
                                        [[0,0,0],[1,0,0,0],[0,-2,1,0],[0,9E+09,9E+09,9E+09,9E+09,9E+09]],
                                        [[0,0,0],[1,0,0,0],[0,-2,1,0],[0,9E+09,9E+09,9E+09,9E+09,9E+09]],
                                        [[0,0,0],[1,0,0,0],[0,-2,1,0],[0,9E+09,9E+09,9E+09,9E+09,9E+09]],
                                        [[0,0,0],[1,0,0,0],[0,-2,1,0],[0,9E+09,9E+09,9E+09,9E+09,9E+09]],
                                        [[0,0,0],[1,0,0,0],[0,-2,1,0],[0,9E+09,9E+09,9E+09,9E+09,9E+09]],
                                        [[0,0,0],[1,0,0,0],[0,-2,1,0],[0,9E+09,9E+09,9E+09,9E+09,9E+09]],
                                        [[0,0,0],[1,0,0,0],[0,-2,1,0],[0,9E+09,9E+09,9E+09,9E+09,9E+09]],
                                        [[0,0,0],[1,0,0,0],[0,-2,1,0],[0,9E+09,9E+09,9E+09,9E+09,9E+09]],
                                        [[0,0,0],[1,0,0,0],[0,-2,1,0],[0,9E+09,9E+09,9E+09,9E+09,9E+09]],
                                        [[0,0,0],[1,0,0,0],[0,-2,1,0],[0,9E+09,9E+09,9E+09,9E+09,9E+09]],
                                        [[0,0,0],[1,0,0,0],[0,-2,1,0],[0,9E+09,9E+09,9E+09,9E+09,9E+09]],
                                        [[0,0,0],[1,0,0,0],[0,-2,1,0],[0,9E+09,9E+09,9E+09,9E+09,9E+09]],
                                        [[0,0,0],[1,0,0,0],[0,-2,1,0],[0,9E+09,9E+09,9E+09,9E+09,9E+09]],
                                        [[0,0,0],[1,0,0,0],[0,-2,1,0],[0,9E+09,9E+09,9E+09,9E+09,9E+09]],
                                        [[0,0,0],[1,0,0,0],[0,-2,1,0],[0,9E+09,9E+09,9E+09,9E+09,9E+09]],
                                        [[0,0,0],[1,0,0,0],[0,-2,1,0],[0,9E+09,9E+09,9E+09,9E+09,9E+09]],
                                        [[0,0,0],[1,0,0,0],[0,-2,1,0],[0,9E+09,9E+09,9E+09,9E+09,9E+09]],
                                        [[0,0,0],[1,0,0,0],[0,-2,1,0],[0,9E+09,9E+09,9E+09,9E+09,9E+09]],
                                        [[0,0,0],[1,0,0,0],[0,-2,1,0],[0,9E+09,9E+09,9E+09,9E+09,9E+09]],
                                        [[0,0,0],[1,0,0,0],[0,-2,1,0],[0,9E+09,9E+09,9E+09,9E+09,9E+09]],
                                        [[0,0,0],[1,0,0,0],[0,-2,1,0],[0,9E+09,9E+09,9E+09,9E+09,9E+09]],
                                        [[0,0,0],[1,0,0,0],[0,-2,1,0],[0,9E+09,9E+09,9E+09,9E+09,9E+09]],
                                        [[0,0,0],[1,0,0,0],[0,-2,1,0],[0,9E+09,9E+09,9E+09,9E+09,9E+09]],
                                        [[0,0,0],[1,0,0,0],[0,-2,1,0],[0,9E+09,9E+09,9E+09,9E+09,9E+09]],
                                        [[0,0,0],[1,0,0,0],[0,-2,1,0],[0,9E+09,9E+09,9E+09,9E+09,9E+09]],
                                        [[0,0,0],[1,0,0,0],[0,-2,1,0],[0,9E+09,9E+09,9E+09,9E+09,9E+09]],
                                        [[0,0,0],[1,0,0,0],[0,-2,1,0],[0,9E+09,9E+09,9E+09,9E+09,9E+09]],
                                        [[0,0,0],[1,0,0,0],[0,-2,1,0],[0,9E+09,9E+09,9E+09,9E+09,9E+09]],
                                        [[0,0,0],[1,0,0,0],[0,-2,1,0],[0,9E+09,9E+09,9E+09,9E+09,9E+09]],
                                        [[0,0,0],[1,0,0,0],[0,-2,1,0],[0,9E+09,9E+09,9E+09,9E+09,9E+09]],
                                        [[0,0,0],[1,0,0,0],[0,-2,1,0],[0,9E+09,9E+09,9E+09,9E+09,9E+09]],
                                        [[0,0,0],[1,0,0,0],[0,-2,1,0],[0,9E+09,9E+09,9E+09,9E+09,9E+09]],
                                        [[0,0,0],[1,0,0,0],[0,-2,1,0],[0,9E+09,9E+09,9E+09,9E+09,9E+09]],
                                        [[0,0,0],[1,0,0,0],[0,-2,1,0],[0,9E+09,9E+09,9E+09,9E+09,9E+09]],
                                        [[0,0,0],[1,0,0,0],[0,-2,1,0],[0,9E+09,9E+09,9E+09,9E+09,9E+09]],
                                        [[0,0,0],[1,0,0,0],[0,-2,1,0],[0,9E+09,9E+09,9E+09,9E+09,9E+09]],
                                        [[0,0,0],[1,0,0,0],[0,-2,1,0],[0,9E+09,9E+09,9E+09,9E+09,9E+09]],
                                        [[0,0,0],[1,0,0,0],[0,-2,1,0],[0,9E+09,9E+09,9E+09,9E+09,9E+09]],
                                        [[0,0,0],[1,0,0,0],[0,-2,1,0],[0,9E+09,9E+09,9E+09,9E+09,9E+09]],
                                        [[0,0,0],[1,0,0,0],[0,-2,1,0],[0,9E+09,9E+09,9E+09,9E+09,9E+09]],
                                        [[0,0,0],[1,0,0,0],[0,-2,1,0],[0,9E+09,9E+09,9E+09,9E+09,9E+09]],
                                        [[0,0,0],[1,0,0,0],[0,-2,1,0],[0,9E+09,9E+09,9E+09,9E+09,9E+09]],
                                        [[0,0,0],[1,0,0,0],[0,-2,1,0],[0,9E+09,9E+09,9E+09,9E+09,9E+09]],
                                        [[0,0,0],[1,0,0,0],[0,-2,1,0],[0,9E+09,9E+09,9E+09,9E+09,9E+09]],
                                        [[0,0,0],[1,0,0,0],[0,-2,1,0],[0,9E+09,9E+09,9E+09,9E+09,9E+09]],
                                        [[0,0,0],[1,0,0,0],[0,-2,1,0],[0,9E+09,9E+09,9E+09,9E+09,9E+09]],
                                        [[0,0,0],[1,0,0,0],[0,-2,1,0],[0,9E+09,9E+09,9E+09,9E+09,9E+09]],
                                        [[0,0,0],[1,0,0,0],[0,-2,1,0],[0,9E+09,9E+09,9E+09,9E+09,9E+09]],
                                        [[0,0,0],[1,0,0,0],[0,-2,1,0],[0,9E+09,9E+09,9E+09,9E+09,9E+09]],
                                        [[0,0,0],[1,0,0,0],[0,-2,1,0],[0,9E+09,9E+09,9E+09,9E+09,9E+09]],
                                        [[0,0,0],[1,0,0,0],[0,-2,1,0],[0,9E+09,9E+09,9E+09,9E+09,9E+09]],
                                        [[0,0,0],[1,0,0,0],[0,-2,1,0],[0,9E+09,9E+09,9E+09,9E+09,9E+09]],
                                        [[0,0,0],[1,0,0,0],[0,-2,1,0],[0,9E+09,9E+09,9E+09,9E+09,9E+09]],
                                        [[0,0,0],[1,0,0,0],[0,-2,1,0],[0,9E+09,9E+09,9E+09,9E+09,9E+09]],
                                        [[0,0,0],[1,0,0,0],[0,-2,1,0],[0,9E+09,9E+09,9E+09,9E+09,9E+09]],
                                        [[0,0,0],[1,0,0,0],[0,-2,1,0],[0,9E+09,9E+09,9E+09,9E+09,9E+09]],
                                        [[0,0,0],[1,0,0,0],[0,-2,1,0],[0,9E+09,9E+09,9E+09,9E+09,9E+09]],
                                        [[0,0,0],[1,0,0,0],[0,-2,1,0],[0,9E+09,9E+09,9E+09,9E+09,9E+09]],
                                        [[0,0,0],[1,0,0,0],[0,-2,1,0],[0,9E+09,9E+09,9E+09,9E+09,9E+09]],
                                        [[0,0,0],[1,0,0,0],[0,-2,1,0],[0,9E+09,9E+09,9E+09,9E+09,9E+09]],
                                        [[0,0,0],[1,0,0,0],[0,-2,1,0],[0,9E+09,9E+09,9E+09,9E+09,9E+09]],
                                        [[0,0,0],[1,0,0,0],[0,-2,1,0],[0,9E+09,9E+09,9E+09,9E+09,9E+09]],
                                        [[0,0,0],[1,0,0,0],[0,-2,1,0],[0,9E+09,9E+09,9E+09,9E+09,9E+09]],
                                        [[0,0,0],[1,0,0,0],[0,-2,1,0],[0,9E+09,9E+09,9E+09,9E+09,9E+09]],
                                        [[0,0,0],[1,0,0,0],[0,-2,1,0],[0,9E+09,9E+09,9E+09,9E+09,9E+09]],
                                        [[0,0,0],[1,0,0,0],[0,-2,1,0],[0,9E+09,9E+09,9E+09,9E+09,9E+09]],
                                        [[0,0,0],[1,0,0,0],[0,-2,1,0],[0,9E+09,9E+09,9E+09,9E+09,9E+09]],
                                        [[0,0,0],[1,0,0,0],[0,-2,1,0],[0,9E+09,9E+09,9E+09,9E+09,9E+09]],
                                        [[0,0,0],[1,0,0,0],[0,-2,1,0],[0,9E+09,9E+09,9E+09,9E+09,9E+09]],
                                        [[0,0,0],[1,0,0,0],[0,-2,1,0],[0,9E+09,9E+09,9E+09,9E+09,9E+09]],
                                        [[0,0,0],[1,0,0,0],[0,-2,1,0],[0,9E+09,9E+09,9E+09,9E+09,9E+09]],
                                        [[0,0,0],[1,0,0,0],[0,-2,1,0],[0,9E+09,9E+09,9E+09,9E+09,9E+09]],
                                        [[0,0,0],[1,0,0,0],[0,-2,1,0],[0,9E+09,9E+09,9E+09,9E+09,9E+09]],
                                        [[0,0,0],[1,0,0,0],[0,-2,1,0],[0,9E+09,9E+09,9E+09,9E+09,9E+09]],
                                        [[0,0,0],[1,0,0,0],[0,-2,1,0],[0,9E+09,9E+09,9E+09,9E+09,9E+09]],
                                        [[0,0,0],[1,0,0,0],[0,-2,1,0],[0,9E+09,9E+09,9E+09,9E+09,9E+09]],
                                        [[0,0,0],[1,0,0,0],[0,-2,1,0],[0,9E+09,9E+09,9E+09,9E+09,9E+09]],
                                        [[0,0,0],[1,0,0,0],[0,-2,1,0],[0,9E+09,9E+09,9E+09,9E+09,9E+09]],
                                        [[0,0,0],[1,0,0,0],[0,-2,1,0],[0,9E+09,9E+09,9E+09,9E+09,9E+09]],
                                        [[0,0,0],[1,0,0,0],[0,-2,1,0],[0,9E+09,9E+09,9E+09,9E+09,9E+09]],
                                        [[0,0,0],[1,0,0,0],[0,-2,1,0],[0,9E+09,9E+09,9E+09,9E+09,9E+09]],
                                        [[0,0,0],[1,0,0,0],[0,-2,1,0],[0,9E+09,9E+09,9E+09,9E+09,9E+09]],
                                        [[0,0,0],[1,0,0,0],[0,-2,1,0],[0,9E+09,9E+09,9E+09,9E+09,9E+09]],
                                        [[0,0,0],[1,0,0,0],[0,-2,1,0],[0,9E+09,9E+09,9E+09,9E+09,9E+09]],
                                        [[0,0,0],[1,0,0,0],[0,-2,1,0],[0,9E+09,9E+09,9E+09,9E+09,9E+09]],
                                        [[0,0,0],[1,0,0,0],[0,-2,1,0],[0,9E+09,9E+09,9E+09,9E+09,9E+09]],
                                        [[0,0,0],[1,0,0,0],[0,-2,1,0],[0,9E+09,9E+09,9E+09,9E+09,9E+09]],
                                        [[0,0,0],[1,0,0,0],[0,-2,1,0],[0,9E+09,9E+09,9E+09,9E+09,9E+09]],
                                        [[0,0,0],[1,0,0,0],[0,-2,1,0],[0,9E+09,9E+09,9E+09,9E+09,9E+09]],
                                        [[0,0,0],[1,0,0,0],[0,-2,1,0],[0,9E+09,9E+09,9E+09,9E+09,9E+09]],
                                        [[0,0,0],[1,0,0,0],[0,-2,1,0],[0,9E+09,9E+09,9E+09,9E+09,9E+09]],
                                        [[0,0,0],[1,0,0,0],[0,-2,1,0],[0,9E+09,9E+09,9E+09,9E+09,9E+09]],
                                        [[0,0,0],[1,0,0,0],[0,-2,1,0],[0,9E+09,9E+09,9E+09,9E+09,9E+09]],
                                        [[0,0,0],[1,0,0,0],[0,-2,1,0],[0,9E+09,9E+09,9E+09,9E+09,9E+09]],
                                        [[0,0,0],[1,0,0,0],[0,-2,1,0],[0,9E+09,9E+09,9E+09,9E+09,9E+09]],
                                        [[0,0,0],[1,0,0,0],[0,-2,1,0],[0,9E+09,9E+09,9E+09,9E+09,9E+09]],
                                        [[0,0,0],[1,0,0,0],[0,-2,1,0],[0,9E+09,9E+09,9E+09,9E+09,9E+09]],
                                        [[0,0,0],[1,0,0,0],[0,-2,1,0],[0,9E+09,9E+09,9E+09,9E+09,9E+09]],
                                        [[0,0,0],[1,0,0,0],[0,-2,1,0],[0,9E+09,9E+09,9E+09,9E+09,9E+09]],
                                        [[0,0,0],[1,0,0,0],[0,-2,1,0],[0,9E+09,9E+09,9E+09,9E+09,9E+09]],
                                        [[0,0,0],[1,0,0,0],[0,-2,1,0],[0,9E+09,9E+09,9E+09,9E+09,9E+09]],
                                        [[0,0,0],[1,0,0,0],[0,-2,1,0],[0,9E+09,9E+09,9E+09,9E+09,9E+09]],
                                        [[0,0,0],[1,0,0,0],[0,-2,1,0],[0,9E+09,9E+09,9E+09,9E+09,9E+09]],
                                        [[0,0,0],[1,0,0,0],[0,-2,1,0],[0,9E+09,9E+09,9E+09,9E+09,9E+09]],
                                        [[0,0,0],[1,0,0,0],[0,-2,1,0],[0,9E+09,9E+09,9E+09,9E+09,9E+09]],
                                        [[0,0,0],[1,0,0,0],[0,-2,1,0],[0,9E+09,9E+09,9E+09,9E+09,9E+09]],
                                        [[0,0,0],[1,0,0,0],[0,-2,1,0],[0,9E+09,9E+09,9E+09,9E+09,9E+09]],
                                        [[0,0,0],[1,0,0,0],[0,-2,1,0],[0,9E+09,9E+09,9E+09,9E+09,9E+09]],
                                        [[0,0,0],[1,0,0,0],[0,-2,1,0],[0,9E+09,9E+09,9E+09,9E+09,9E+09]],
                                        [[0,0,0],[1,0,0,0],[0,-2,1,0],[0,9E+09,9E+09,9E+09,9E+09,9E+09]],
                                        [[0,0,0],[1,0,0,0],[0,-2,1,0],[0,9E+09,9E+09,9E+09,9E+09,9E+09]],
                                        [[0,0,0],[1,0,0,0],[0,-2,1,0],[0,9E+09,9E+09,9E+09,9E+09,9E+09]],
                                        [[0,0,0],[1,0,0,0],[0,-2,1,0],[0,9E+09,9E+09,9E+09,9E+09,9E+09]],
                                        [[0,0,0],[1,0,0,0],[0,-2,1,0],[0,9E+09,9E+09,9E+09,9E+09,9E+09]],
                                        [[0,0,0],[1,0,0,0],[0,-2,1,0],[0,9E+09,9E+09,9E+09,9E+09,9E+09]],
                                        [[0,0,0],[1,0,0,0],[0,-2,1,0],[0,9E+09,9E+09,9E+09,9E+09,9E+09]],
                                        [[0,0,0],[1,0,0,0],[0,-2,1,0],[0,9E+09,9E+09,9E+09,9E+09,9E+09]],
                                        [[0,0,0],[1,0,0,0],[0,-2,1,0],[0,9E+09,9E+09,9E+09,9E+09,9E+09]],
                                        [[0,0,0],[1,0,0,0],[0,-2,1,0],[0,9E+09,9E+09,9E+09,9E+09,9E+09]],
                                        [[0,0,0],[1,0,0,0],[0,-2,1,0],[0,9E+09,9E+09,9E+09,9E+09,9E+09]],
                                        [[0,0,0],[1,0,0,0],[0,-2,1,0],[0,9E+09,9E+09,9E+09,9E+09,9E+09]],
                                        [[0,0,0],[1,0,0,0],[0,-2,1,0],[0,9E+09,9E+09,9E+09,9E+09,9E+09]],
                                        [[0,0,0],[1,0,0,0],[0,-2,1,0],[0,9E+09,9E+09,9E+09,9E+09,9E+09]],
                                        [[0,0,0],[1,0,0,0],[0,-2,1,0],[0,9E+09,9E+09,9E+09,9E+09,9E+09]],
                                        [[0,0,0],[1,0,0,0],[0,-2,1,0],[0,9E+09,9E+09,9E+09,9E+09,9E+09]],
                                        [[0,0,0],[1,0,0,0],[0,-2,1,0],[0,9E+09,9E+09,9E+09,9E+09,9E+09]],
                                        [[0,0,0],[1,0,0,0],[0,-2,1,0],[0,9E+09,9E+09,9E+09,9E+09,9E+09]],
                                        [[0,0,0],[1,0,0,0],[0,-2,1,0],[0,9E+09,9E+09,9E+09,9E+09,9E+09]],
                                        [[0,0,0],[1,0,0,0],[0,-2,1,0],[0,9E+09,9E+09,9E+09,9E+09,9E+09]],
                                        [[0,0,0],[1,0,0,0],[0,-2,1,0],[0,9E+09,9E+09,9E+09,9E+09,9E+09]],
                                        [[0,0,0],[1,0,0,0],[0,-2,1,0],[0,9E+09,9E+09,9E+09,9E+09,9E+09]],
                                        [[0,0,0],[1,0,0,0],[0,-2,1,0],[0,9E+09,9E+09,9E+09,9E+09,9E+09]],
                                        [[0,0,0],[1,0,0,0],[0,-2,1,0],[0,9E+09,9E+09,9E+09,9E+09,9E+09]],
                                        [[0,0,0],[1,0,0,0],[0,-2,1,0],[0,9E+09,9E+09,9E+09,9E+09,9E+09]],
                                        [[0,0,0],[1,0,0,0],[0,-2,1,0],[0,9E+09,9E+09,9E+09,9E+09,9E+09]],
                                        [[0,0,0],[1,0,0,0],[0,-2,1,0],[0,9E+09,9E+09,9E+09,9E+09,9E+09]],
                                        [[0,0,0],[1,0,0,0],[0,-2,1,0],[0,9E+09,9E+09,9E+09,9E+09,9E+09]],
                                        [[0,0,0],[1,0,0,0],[0,-2,1,0],[0,9E+09,9E+09,9E+09,9E+09,9E+09]],
                                        [[0,0,0],[1,0,0,0],[0,-2,1,0],[0,9E+09,9E+09,9E+09,9E+09,9E+09]],
                                        [[0,0,0],[1,0,0,0],[0,-2,1,0],[0,9E+09,9E+09,9E+09,9E+09,9E+09]],
                                        [[0,0,0],[1,0,0,0],[0,-2,1,0],[0,9E+09,9E+09,9E+09,9E+09,9E+09]],
                                        [[0,0,0],[1,0,0,0],[0,-2,1,0],[0,9E+09,9E+09,9E+09,9E+09,9E+09]],
                                        [[0,0,0],[1,0,0,0],[0,-2,1,0],[0,9E+09,9E+09,9E+09,9E+09,9E+09]],
                                        [[0,0,0],[1,0,0,0],[0,-2,1,0],[0,9E+09,9E+09,9E+09,9E+09,9E+09]],
                                        [[0,0,0],[1,0,0,0],[0,-2,1,0],[0,9E+09,9E+09,9E+09,9E+09,9E+09]],
                                        [[0,0,0],[1,0,0,0],[0,-2,1,0],[0,9E+09,9E+09,9E+09,9E+09,9E+09]],
                                        [[0,0,0],[1,0,0,0],[0,-2,1,0],[0,9E+09,9E+09,9E+09,9E+09,9E+09]],
                                        [[0,0,0],[1,0,0,0],[0,-2,1,0],[0,9E+09,9E+09,9E+09,9E+09,9E+09]],
                                        [[0,0,0],[1,0,0,0],[0,-2,1,0],[0,9E+09,9E+09,9E+09,9E+09,9E+09]],
                                        [[0,0,0],[1,0,0,0],[0,-2,1,0],[0,9E+09,9E+09,9E+09,9E+09,9E+09]],
                                        [[0,0,0],[1,0,0,0],[0,-2,1,0],[0,9E+09,9E+09,9E+09,9E+09,9E+09]],
                                        [[0,0,0],[1,0,0,0],[0,-2,1,0],[0,9E+09,9E+09,9E+09,9E+09,9E+09]],
                                        [[0,0,0],[1,0,0,0],[0,-2,1,0],[0,9E+09,9E+09,9E+09,9E+09,9E+09]],
                                        [[0,0,0],[1,0,0,0],[0,-2,1,0],[0,9E+09,9E+09,9E+09,9E+09,9E+09]],
                                        [[0,0,0],[1,0,0,0],[0,-2,1,0],[0,9E+09,9E+09,9E+09,9E+09,9E+09]],
                                        [[0,0,0],[1,0,0,0],[0,-2,1,0],[0,9E+09,9E+09,9E+09,9E+09,9E+09]],
                                        [[0,0,0],[1,0,0,0],[0,-2,1,0],[0,9E+09,9E+09,9E+09,9E+09,9E+09]],
                                        [[0,0,0],[1,0,0,0],[0,-2,1,0],[0,9E+09,9E+09,9E+09,9E+09,9E+09]],
                                        [[0,0,0],[1,0,0,0],[0,-2,1,0],[0,9E+09,9E+09,9E+09,9E+09,9E+09]],
                                        [[0,0,0],[1,0,0,0],[0,-2,1,0],[0,9E+09,9E+09,9E+09,9E+09,9E+09]],
                                        [[0,0,0],[1,0,0,0],[0,-2,1,0],[0,9E+09,9E+09,9E+09,9E+09,9E+09]],
                                        [[0,0,0],[1,0,0,0],[0,-2,1,0],[0,9E+09,9E+09,9E+09,9E+09,9E+09]],
                                        [[0,0,0],[1,0,0,0],[0,-2,1,0],[0,9E+09,9E+09,9E+09,9E+09,9E+09]],
                                        [[0,0,0],[1,0,0,0],[0,-2,1,0],[0,9E+09,9E+09,9E+09,9E+09,9E+09]],
                                        [[0,0,0],[1,0,0,0],[0,-2,1,0],[0,9E+09,9E+09,9E+09,9E+09,9E+09]],
                                        [[0,0,0],[1,0,0,0],[0,-2,1,0],[0,9E+09,9E+09,9E+09,9E+09,9E+09]],
                                        [[0,0,0],[1,0,0,0],[0,-2,1,0],[0,9E+09,9E+09,9E+09,9E+09,9E+09]],
                                        [[0,0,0],[1,0,0,0],[0,-2,1,0],[0,9E+09,9E+09,9E+09,9E+09,9E+09]],
                                        [[0,0,0],[1,0,0,0],[0,-2,1,0],[0,9E+09,9E+09,9E+09,9E+09,9E+09]],
                                        [[0,0,0],[1,0,0,0],[0,-2,1,0],[0,9E+09,9E+09,9E+09,9E+09,9E+09]],
                                        [[0,0,0],[1,0,0,0],[0,-2,1,0],[0,9E+09,9E+09,9E+09,9E+09,9E+09]],
                                        [[0,0,0],[1,0,0,0],[0,-2,1,0],[0,9E+09,9E+09,9E+09,9E+09,9E+09]],
                                        [[0,0,0],[1,0,0,0],[0,-2,1,0],[0,9E+09,9E+09,9E+09,9E+09,9E+09]],
                                        [[0,0,0],[1,0,0,0],[0,-2,1,0],[0,9E+09,9E+09,9E+09,9E+09,9E+09]],
                                        [[0,0,0],[1,0,0,0],[0,-2,1,0],[0,9E+09,9E+09,9E+09,9E+09,9E+09]],
                                        [[0,0,0],[1,0,0,0],[0,-2,1,0],[0,9E+09,9E+09,9E+09,9E+09,9E+09]],
                                        [[0,0,0],[1,0,0,0],[0,-2,1,0],[0,9E+09,9E+09,9E+09,9E+09,9E+09]],
                                        [[0,0,0],[1,0,0,0],[0,-2,1,0],[0,9E+09,9E+09,9E+09,9E+09,9E+09]],
                                        [[0,0,0],[1,0,0,0],[0,-2,1,0],[0,9E+09,9E+09,9E+09,9E+09,9E+09]],
                                        [[0,0,0],[1,0,0,0],[0,-2,1,0],[0,9E+09,9E+09,9E+09,9E+09,9E+09]],
                                        [[0,0,0],[1,0,0,0],[0,-2,1,0],[0,9E+09,9E+09,9E+09,9E+09,9E+09]],
                                        [[0,0,0],[1,0,0,0],[0,-2,1,0],[0,9E+09,9E+09,9E+09,9E+09,9E+09]],
                                        [[0,0,0],[1,0,0,0],[0,-2,1,0],[0,9E+09,9E+09,9E+09,9E+09,9E+09]],
                                        [[0,0,0],[1,0,0,0],[0,-2,1,0],[0,9E+09,9E+09,9E+09,9E+09,9E+09]],
                                        [[0,0,0],[1,0,0,0],[0,-2,1,0],[0,9E+09,9E+09,9E+09,9E+09,9E+09]],
                                        [[0,0,0],[1,0,0,0],[0,-2,1,0],[0,9E+09,9E+09,9E+09,9E+09,9E+09]],
                                        [[0,0,0],[1,0,0,0],[0,-2,1,0],[0,9E+09,9E+09,9E+09,9E+09,9E+09]],
                                        [[0,0,0],[1,0,0,0],[0,-2,1,0],[0,9E+09,9E+09,9E+09,9E+09,9E+09]],
                                        [[0,0,0],[1,0,0,0],[0,-2,1,0],[0,9E+09,9E+09,9E+09,9E+09,9E+09]],
                                        [[0,0,0],[1,0,0,0],[0,-2,1,0],[0,9E+09,9E+09,9E+09,9E+09,9E+09]],
                                        [[0,0,0],[1,0,0,0],[0,-2,1,0],[0,9E+09,9E+09,9E+09,9E+09,9E+09]],
                                        [[0,0,0],[1,0,0,0],[0,-2,1,0],[0,9E+09,9E+09,9E+09,9E+09,9E+09]],
                                        [[0,0,0],[1,0,0,0],[0,-2,1,0],[0,9E+09,9E+09,9E+09,9E+09,9E+09]],
                                        [[0,0,0],[1,0,0,0],[0,-2,1,0],[0,9E+09,9E+09,9E+09,9E+09,9E+09]],
                                        [[0,0,0],[1,0,0,0],[0,-2,1,0],[0,9E+09,9E+09,9E+09,9E+09,9E+09]],
                                        [[0,0,0],[1,0,0,0],[0,-2,1,0],[0,9E+09,9E+09,9E+09,9E+09,9E+09]],
                                        [[0,0,0],[1,0,0,0],[0,-2,1,0],[0,9E+09,9E+09,9E+09,9E+09,9E+09]],
                                        [[0,0,0],[1,0,0,0],[0,-2,1,0],[0,9E+09,9E+09,9E+09,9E+09,9E+09]],
                                        [[0,0,0],[1,0,0,0],[0,-2,1,0],[0,9E+09,9E+09,9E+09,9E+09,9E+09]],
                                        [[0,0,0],[1,0,0,0],[0,-2,1,0],[0,9E+09,9E+09,9E+09,9E+09,9E+09]],
                                        [[0,0,0],[1,0,0,0],[0,-2,1,0],[0,9E+09,9E+09,9E+09,9E+09,9E+09]],
                                        [[0,0,0],[1,0,0,0],[0,-2,1,0],[0,9E+09,9E+09,9E+09,9E+09,9E+09]],
                                        [[0,0,0],[1,0,0,0],[0,-2,1,0],[0,9E+09,9E+09,9E+09,9E+09,9E+09]],
                                        [[0,0,0],[1,0,0,0],[0,-2,1,0],[0,9E+09,9E+09,9E+09,9E+09,9E+09]],
                                        [[0,0,0],[1,0,0,0],[0,-2,1,0],[0,9E+09,9E+09,9E+09,9E+09,9E+09]],
                                        [[0,0,0],[1,0,0,0],[0,-2,1,0],[0,9E+09,9E+09,9E+09,9E+09,9E+09]],
                                        [[0,0,0],[1,0,0,0],[0,-2,1,0],[0,9E+09,9E+09,9E+09,9E+09,9E+09]],
                                        [[0,0,0],[1,0,0,0],[0,-2,1,0],[0,9E+09,9E+09,9E+09,9E+09,9E+09]],
                                        [[0,0,0],[1,0,0,0],[0,-2,1,0],[0,9E+09,9E+09,9E+09,9E+09,9E+09]],
                                        [[0,0,0],[1,0,0,0],[0,-2,1,0],[0,9E+09,9E+09,9E+09,9E+09,9E+09]],
                                        [[0,0,0],[1,0,0,0],[0,-2,1,0],[0,9E+09,9E+09,9E+09,9E+09,9E+09]],
                                        [[0,0,0],[1,0,0,0],[0,-2,1,0],[0,9E+09,9E+09,9E+09,9E+09,9E+09]],
                                        [[0,0,0],[1,0,0,0],[0,-2,1,0],[0,9E+09,9E+09,9E+09,9E+09,9E+09]],
                                        [[0,0,0],[1,0,0,0],[0,-2,1,0],[0,9E+09,9E+09,9E+09,9E+09,9E+09]],
                                        [[0,0,0],[1,0,0,0],[0,-2,1,0],[0,9E+09,9E+09,9E+09,9E+09,9E+09]],
                                        [[0,0,0],[1,0,0,0],[0,-2,1,0],[0,9E+09,9E+09,9E+09,9E+09,9E+09]],
                                        [[0,0,0],[1,0,0,0],[0,-2,1,0],[0,9E+09,9E+09,9E+09,9E+09,9E+09]],
                                        [[0,0,0],[1,0,0,0],[0,-2,1,0],[0,9E+09,9E+09,9E+09,9E+09,9E+09]],
                                        [[0,0,0],[1,0,0,0],[0,-2,1,0],[0,9E+09,9E+09,9E+09,9E+09,9E+09]],
                                        [[0,0,0],[1,0,0,0],[0,-2,1,0],[0,9E+09,9E+09,9E+09,9E+09,9E+09]],
                                        [[0,0,0],[1,0,0,0],[0,-2,1,0],[0,9E+09,9E+09,9E+09,9E+09,9E+09]],
                                        [[0,0,0],[1,0,0,0],[0,-2,1,0],[0,9E+09,9E+09,9E+09,9E+09,9E+09]],
                                        [[0,0,0],[1,0,0,0],[0,-2,1,0],[0,9E+09,9E+09,9E+09,9E+09,9E+09]],
                                        [[0,0,0],[1,0,0,0],[0,-2,1,0],[0,9E+09,9E+09,9E+09,9E+09,9E+09]],
                                        [[0,0,0],[1,0,0,0],[0,-2,1,0],[0,9E+09,9E+09,9E+09,9E+09,9E+09]],
                                        [[0,0,0],[1,0,0,0],[0,-2,1,0],[0,9E+09,9E+09,9E+09,9E+09,9E+09]],
                                        [[0,0,0],[1,0,0,0],[0,-2,1,0],[0,9E+09,9E+09,9E+09,9E+09,9E+09]],
                                        [[0,0,0],[1,0,0,0],[0,-2,1,0],[0,9E+09,9E+09,9E+09,9E+09,9E+09]],
                                        [[0,0,0],[1,0,0,0],[0,-2,1,0],[0,9E+09,9E+09,9E+09,9E+09,9E+09]],
                                        [[0,0,0],[1,0,0,0],[0,-2,1,0],[0,9E+09,9E+09,9E+09,9E+09,9E+09]],
                                        [[0,0,0],[1,0,0,0],[0,-2,1,0],[0,9E+09,9E+09,9E+09,9E+09,9E+09]],
                                        [[0,0,0],[1,0,0,0],[0,-2,1,0],[0,9E+09,9E+09,9E+09,9E+09,9E+09]],
                                        [[0,0,0],[1,0,0,0],[0,-2,1,0],[0,9E+09,9E+09,9E+09,9E+09,9E+09]],
                                        [[0,0,0],[1,0,0,0],[0,-2,1,0],[0,9E+09,9E+09,9E+09,9E+09,9E+09]],
                                        [[0,0,0],[1,0,0,0],[0,-2,1,0],[0,9E+09,9E+09,9E+09,9E+09,9E+09]],
                                        [[0,0,0],[1,0,0,0],[0,-2,1,0],[0,9E+09,9E+09,9E+09,9E+09,9E+09]],
                                        [[0,0,0],[1,0,0,0],[0,-2,1,0],[0,9E+09,9E+09,9E+09,9E+09,9E+09]],
                                        [[0,0,0],[1,0,0,0],[0,-2,1,0],[0,9E+09,9E+09,9E+09,9E+09,9E+09]],
                                        [[0,0,0],[1,0,0,0],[0,-2,1,0],[0,9E+09,9E+09,9E+09,9E+09,9E+09]],
                                        [[0,0,0],[1,0,0,0],[0,-2,1,0],[0,9E+09,9E+09,9E+09,9E+09,9E+09]],
                                        [[0,0,0],[1,0,0,0],[0,-2,1,0],[0,9E+09,9E+09,9E+09,9E+09,9E+09]],
                                        [[0,0,0],[1,0,0,0],[0,-2,1,0],[0,9E+09,9E+09,9E+09,9E+09,9E+09]],
                                        [[0,0,0],[1,0,0,0],[0,-2,1,0],[0,9E+09,9E+09,9E+09,9E+09,9E+09]],
                                        [[0,0,0],[1,0,0,0],[0,-2,1,0],[0,9E+09,9E+09,9E+09,9E+09,9E+09]],
                                        [[0,0,0],[1,0,0,0],[0,-2,1,0],[0,9E+09,9E+09,9E+09,9E+09,9E+09]],
                                        [[0,0,0],[1,0,0,0],[0,-2,1,0],[0,9E+09,9E+09,9E+09,9E+09,9E+09]],
                                        [[0,0,0],[1,0,0,0],[0,-2,1,0],[0,9E+09,9E+09,9E+09,9E+09,9E+09]],
                                        [[0,0,0],[1,0,0,0],[0,-2,1,0],[0,9E+09,9E+09,9E+09,9E+09,9E+09]],
                                        [[0,0,0],[1,0,0,0],[0,-2,1,0],[0,9E+09,9E+09,9E+09,9E+09,9E+09]],
                                        [[0,0,0],[1,0,0,0],[0,-2,1,0],[0,9E+09,9E+09,9E+09,9E+09,9E+09]],
                                        [[0,0,0],[1,0,0,0],[0,-2,1,0],[0,9E+09,9E+09,9E+09,9E+09,9E+09]],
                                        [[0,0,0],[1,0,0,0],[0,-2,1,0],[0,9E+09,9E+09,9E+09,9E+09,9E+09]],
                                        [[0,0,0],[1,0,0,0],[0,-2,1,0],[0,9E+09,9E+09,9E+09,9E+09,9E+09]],
                                        [[0,0,0],[1,0,0,0],[0,-2,1,0],[0,9E+09,9E+09,9E+09,9E+09,9E+09]],
                                        [[0,0,0],[1,0,0,0],[0,-2,1,0],[0,9E+09,9E+09,9E+09,9E+09,9E+09]],
                                        [[0,0,0],[1,0,0,0],[0,-2,1,0],[0,9E+09,9E+09,9E+09,9E+09,9E+09]],
                                        [[0,0,0],[1,0,0,0],[0,-2,1,0],[0,9E+09,9E+09,9E+09,9E+09,9E+09]],
                                        [[0,0,0],[1,0,0,0],[0,-2,1,0],[0,9E+09,9E+09,9E+09,9E+09,9E+09]],
                                        [[0,0,0],[1,0,0,0],[0,-2,1,0],[0,9E+09,9E+09,9E+09,9E+09,9E+09]],
                                        [[0,0,0],[1,0,0,0],[0,-2,1,0],[0,9E+09,9E+09,9E+09,9E+09,9E+09]],
                                        [[0,0,0],[1,0,0,0],[0,-2,1,0],[0,9E+09,9E+09,9E+09,9E+09,9E+09]],
                                        [[0,0,0],[1,0,0,0],[0,-2,1,0],[0,9E+09,9E+09,9E+09,9E+09,9E+09]],
                                        [[0,0,0],[1,0,0,0],[0,-2,1,0],[0,9E+09,9E+09,9E+09,9E+09,9E+09]],
                                        [[0,0,0],[1,0,0,0],[0,-2,1,0],[0,9E+09,9E+09,9E+09,9E+09,9E+09]],
                                        [[0,0,0],[1,0,0,0],[0,-2,1,0],[0,9E+09,9E+09,9E+09,9E+09,9E+09]],
                                        [[0,0,0],[1,0,0,0],[0,-2,1,0],[0,9E+09,9E+09,9E+09,9E+09,9E+09]],
                                        [[0,0,0],[1,0,0,0],[0,-2,1,0],[0,9E+09,9E+09,9E+09,9E+09,9E+09]],
                                        [[0,0,0],[1,0,0,0],[0,-2,1,0],[0,9E+09,9E+09,9E+09,9E+09,9E+09]],
                                        [[0,0,0],[1,0,0,0],[0,-2,1,0],[0,9E+09,9E+09,9E+09,9E+09,9E+09]],
                                        [[0,0,0],[1,0,0,0],[0,-2,1,0],[0,9E+09,9E+09,9E+09,9E+09,9E+09]],
                                        [[0,0,0],[1,0,0,0],[0,-2,1,0],[0,9E+09,9E+09,9E+09,9E+09,9E+09]],
                                        [[0,0,0],[1,0,0,0],[0,-2,1,0],[0,9E+09,9E+09,9E+09,9E+09,9E+09]],
                                        [[0,0,0],[1,0,0,0],[0,-2,1,0],[0,9E+09,9E+09,9E+09,9E+09,9E+09]],
                                        [[0,0,0],[1,0,0,0],[0,-2,1,0],[0,9E+09,9E+09,9E+09,9E+09,9E+09]],
                                        [[0,0,0],[1,0,0,0],[0,-2,1,0],[0,9E+09,9E+09,9E+09,9E+09,9E+09]],
                                        [[0,0,0],[1,0,0,0],[0,-2,1,0],[0,9E+09,9E+09,9E+09,9E+09,9E+09]],
                                        [[0,0,0],[1,0,0,0],[0,-2,1,0],[0,9E+09,9E+09,9E+09,9E+09,9E+09]],
                                        [[0,0,0],[1,0,0,0],[0,-2,1,0],[0,9E+09,9E+09,9E+09,9E+09,9E+09]],
                                        [[0,0,0],[1,0,0,0],[0,-2,1,0],[0,9E+09,9E+09,9E+09,9E+09,9E+09]],
                                        [[0,0,0],[1,0,0,0],[0,-2,1,0],[0,9E+09,9E+09,9E+09,9E+09,9E+09]],
                                        [[0,0,0],[1,0,0,0],[0,-2,1,0],[0,9E+09,9E+09,9E+09,9E+09,9E+09]],
                                        [[0,0,0],[1,0,0,0],[0,-2,1,0],[0,9E+09,9E+09,9E+09,9E+09,9E+09]],
                                        [[0,0,0],[1,0,0,0],[0,-2,1,0],[0,9E+09,9E+09,9E+09,9E+09,9E+09]],
                                        [[0,0,0],[1,0,0,0],[0,-2,1,0],[0,9E+09,9E+09,9E+09,9E+09,9E+09]],
                                        [[0,0,0],[1,0,0,0],[0,-2,1,0],[0,9E+09,9E+09,9E+09,9E+09,9E+09]],
                                        [[0,0,0],[1,0,0,0],[0,-2,1,0],[0,9E+09,9E+09,9E+09,9E+09,9E+09]],
                                        [[0,0,0],[1,0,0,0],[0,-2,1,0],[0,9E+09,9E+09,9E+09,9E+09,9E+09]],
                                        [[0,0,0],[1,0,0,0],[0,-2,1,0],[0,9E+09,9E+09,9E+09,9E+09,9E+09]],
                                        [[0,0,0],[1,0,0,0],[0,-2,1,0],[0,9E+09,9E+09,9E+09,9E+09,9E+09]],
                                        [[0,0,0],[1,0,0,0],[0,-2,1,0],[0,9E+09,9E+09,9E+09,9E+09,9E+09]],
                                        [[0,0,0],[1,0,0,0],[0,-2,1,0],[0,9E+09,9E+09,9E+09,9E+09,9E+09]],
                                        [[0,0,0],[1,0,0,0],[0,-2,1,0],[0,9E+09,9E+09,9E+09,9E+09,9E+09]],
                                        [[0,0,0],[1,0,0,0],[0,-2,1,0],[0,9E+09,9E+09,9E+09,9E+09,9E+09]],
                                        [[0,0,0],[1,0,0,0],[0,-2,1,0],[0,9E+09,9E+09,9E+09,9E+09,9E+09]],
                                        [[0,0,0],[1,0,0,0],[0,-2,1,0],[0,9E+09,9E+09,9E+09,9E+09,9E+09]],
                                        [[0,0,0],[1,0,0,0],[0,-2,1,0],[0,9E+09,9E+09,9E+09,9E+09,9E+09]],
                                        [[0,0,0],[1,0,0,0],[0,-2,1,0],[0,9E+09,9E+09,9E+09,9E+09,9E+09]],
                                        [[0,0,0],[1,0,0,0],[0,-2,1,0],[0,9E+09,9E+09,9E+09,9E+09,9E+09]],
                                        [[0,0,0],[1,0,0,0],[0,-2,1,0],[0,9E+09,9E+09,9E+09,9E+09,9E+09]],
                                        [[0,0,0],[1,0,0,0],[0,-2,1,0],[0,9E+09,9E+09,9E+09,9E+09,9E+09]],
                                        [[0,0,0],[1,0,0,0],[0,-2,1,0],[0,9E+09,9E+09,9E+09,9E+09,9E+09]],
                                        [[0,0,0],[1,0,0,0],[0,-2,1,0],[0,9E+09,9E+09,9E+09,9E+09,9E+09]],
                                        [[0,0,0],[1,0,0,0],[0,-2,1,0],[0,9E+09,9E+09,9E+09,9E+09,9E+09]],
                                        [[0,0,0],[1,0,0,0],[0,-2,1,0],[0,9E+09,9E+09,9E+09,9E+09,9E+09]],
                                        [[0,0,0],[1,0,0,0],[0,-2,1,0],[0,9E+09,9E+09,9E+09,9E+09,9E+09]],
                                        [[0,0,0],[1,0,0,0],[0,-2,1,0],[0,9E+09,9E+09,9E+09,9E+09,9E+09]],
                                        [[0,0,0],[1,0,0,0],[0,-2,1,0],[0,9E+09,9E+09,9E+09,9E+09,9E+09]],
                                        [[0,0,0],[1,0,0,0],[0,-2,1,0],[0,9E+09,9E+09,9E+09,9E+09,9E+09]],
                                        [[0,0,0],[1,0,0,0],[0,-2,1,0],[0,9E+09,9E+09,9E+09,9E+09,9E+09]],
                                        [[0,0,0],[1,0,0,0],[0,-2,1,0],[0,9E+09,9E+09,9E+09,9E+09,9E+09]],
                                        [[0,0,0],[1,0,0,0],[0,-2,1,0],[0,9E+09,9E+09,9E+09,9E+09,9E+09]],
                                        [[0,0,0],[1,0,0,0],[0,-2,1,0],[0,9E+09,9E+09,9E+09,9E+09,9E+09]],
                                        [[0,0,0],[1,0,0,0],[0,-2,1,0],[0,9E+09,9E+09,9E+09,9E+09,9E+09]],
                                        [[0,0,0],[1,0,0,0],[0,-2,1,0],[0,9E+09,9E+09,9E+09,9E+09,9E+09]],
                                        [[0,0,0],[1,0,0,0],[0,-2,1,0],[0,9E+09,9E+09,9E+09,9E+09,9E+09]],
                                        [[0,0,0],[1,0,0,0],[0,-2,1,0],[0,9E+09,9E+09,9E+09,9E+09,9E+09]],
                                        [[0,0,0],[1,0,0,0],[0,-2,1,0],[0,9E+09,9E+09,9E+09,9E+09,9E+09]],
                                        [[0,0,0],[1,0,0,0],[0,-2,1,0],[0,9E+09,9E+09,9E+09,9E+09,9E+09]],
                                        [[0,0,0],[1,0,0,0],[0,-2,1,0],[0,9E+09,9E+09,9E+09,9E+09,9E+09]],
                                        [[0,0,0],[1,0,0,0],[0,-2,1,0],[0,9E+09,9E+09,9E+09,9E+09,9E+09]],
                                        [[0,0,0],[1,0,0,0],[0,-2,1,0],[0,9E+09,9E+09,9E+09,9E+09,9E+09]],
                                        [[0,0,0],[1,0,0,0],[0,-2,1,0],[0,9E+09,9E+09,9E+09,9E+09,9E+09]],
                                        [[0,0,0],[1,0,0,0],[0,-2,1,0],[0,9E+09,9E+09,9E+09,9E+09,9E+09]],
                                        [[0,0,0],[1,0,0,0],[0,-2,1,0],[0,9E+09,9E+09,9E+09,9E+09,9E+09]],
                                        [[0,0,0],[1,0,0,0],[0,-2,1,0],[0,9E+09,9E+09,9E+09,9E+09,9E+09]],
                                        [[0,0,0],[1,0,0,0],[0,-2,1,0],[0,9E+09,9E+09,9E+09,9E+09,9E+09]],
                                        [[0,0,0],[1,0,0,0],[0,-2,1,0],[0,9E+09,9E+09,9E+09,9E+09,9E+09]],
                                        [[0,0,0],[1,0,0,0],[0,-2,1,0],[0,9E+09,9E+09,9E+09,9E+09,9E+09]],
                                        [[0,0,0],[1,0,0,0],[0,-2,1,0],[0,9E+09,9E+09,9E+09,9E+09,9E+09]],
                                        [[0,0,0],[1,0,0,0],[0,-2,1,0],[0,9E+09,9E+09,9E+09,9E+09,9E+09]],
                                        [[0,0,0],[1,0,0,0],[0,-2,1,0],[0,9E+09,9E+09,9E+09,9E+09,9E+09]],
                                        [[0,0,0],[1,0,0,0],[0,-2,1,0],[0,9E+09,9E+09,9E+09,9E+09,9E+09]],
                                        [[0,0,0],[1,0,0,0],[0,-2,1,0],[0,9E+09,9E+09,9E+09,9E+09,9E+09]],
                                        [[0,0,0],[1,0,0,0],[0,-2,1,0],[0,9E+09,9E+09,9E+09,9E+09,9E+09]],
                                        [[0,0,0],[1,0,0,0],[0,-2,1,0],[0,9E+09,9E+09,9E+09,9E+09,9E+09]],
                                        [[0,0,0],[1,0,0,0],[0,-2,1,0],[0,9E+09,9E+09,9E+09,9E+09,9E+09]],
                                        [[0,0,0],[1,0,0,0],[0,-2,1,0],[0,9E+09,9E+09,9E+09,9E+09,9E+09]],
                                        [[0,0,0],[1,0,0,0],[0,-2,1,0],[0,9E+09,9E+09,9E+09,9E+09,9E+09]],
                                        [[0,0,0],[1,0,0,0],[0,-2,1,0],[0,9E+09,9E+09,9E+09,9E+09,9E+09]],
                                        [[0,0,0],[1,0,0,0],[0,-2,1,0],[0,9E+09,9E+09,9E+09,9E+09,9E+09]],
                                        [[0,0,0],[1,0,0,0],[0,-2,1,0],[0,9E+09,9E+09,9E+09,9E+09,9E+09]],
                                        [[0,0,0],[1,0,0,0],[0,-2,1,0],[0,9E+09,9E+09,9E+09,9E+09,9E+09]],
                                        [[0,0,0],[1,0,0,0],[0,-2,1,0],[0,9E+09,9E+09,9E+09,9E+09,9E+09]],
                                        [[0,0,0],[1,0,0,0],[0,-2,1,0],[0,9E+09,9E+09,9E+09,9E+09,9E+09]],
                                        [[0,0,0],[1,0,0,0],[0,-2,1,0],[0,9E+09,9E+09,9E+09,9E+09,9E+09]],
                                        [[0,0,0],[1,0,0,0],[0,-2,1,0],[0,9E+09,9E+09,9E+09,9E+09,9E+09]],
                                        [[0,0,0],[1,0,0,0],[0,-2,1,0],[0,9E+09,9E+09,9E+09,9E+09,9E+09]],
                                        [[0,0,0],[1,0,0,0],[0,-2,1,0],[0,9E+09,9E+09,9E+09,9E+09,9E+09]],
                                        [[0,0,0],[1,0,0,0],[0,-2,1,0],[0,9E+09,9E+09,9E+09,9E+09,9E+09]],
                                        [[0,0,0],[1,0,0,0],[0,-2,1,0],[0,9E+09,9E+09,9E+09,9E+09,9E+09]],
                                        [[0,0,0],[1,0,0,0],[0,-2,1,0],[0,9E+09,9E+09,9E+09,9E+09,9E+09]],
                                        [[0,0,0],[1,0,0,0],[0,-2,1,0],[0,9E+09,9E+09,9E+09,9E+09,9E+09]],
                                        [[0,0,0],[1,0,0,0],[0,-2,1,0],[0,9E+09,9E+09,9E+09,9E+09,9E+09]],
                                        [[0,0,0],[1,0,0,0],[0,-2,1,0],[0,9E+09,9E+09,9E+09,9E+09,9E+09]],
                                        [[0,0,0],[1,0,0,0],[0,-2,1,0],[0,9E+09,9E+09,9E+09,9E+09,9E+09]],
                                        [[0,0,0],[1,0,0,0],[0,-2,1,0],[0,9E+09,9E+09,9E+09,9E+09,9E+09]],
                                        [[0,0,0],[1,0,0,0],[0,-2,1,0],[0,9E+09,9E+09,9E+09,9E+09,9E+09]],
                                        [[0,0,0],[1,0,0,0],[0,-2,1,0],[0,9E+09,9E+09,9E+09,9E+09,9E+09]],
                                        [[0,0,0],[1,0,0,0],[0,-2,1,0],[0,9E+09,9E+09,9E+09,9E+09,9E+09]],
                                        [[0,0,0],[1,0,0,0],[0,-2,1,0],[0,9E+09,9E+09,9E+09,9E+09,9E+09]],
                                        [[0,0,0],[1,0,0,0],[0,-2,1,0],[0,9E+09,9E+09,9E+09,9E+09,9E+09]],
                                        [[0,0,0],[1,0,0,0],[0,-2,1,0],[0,9E+09,9E+09,9E+09,9E+09,9E+09]],
                                        [[0,0,0],[1,0,0,0],[0,-2,1,0],[0,9E+09,9E+09,9E+09,9E+09,9E+09]],
                                        [[0,0,0],[1,0,0,0],[0,-2,1,0],[0,9E+09,9E+09,9E+09,9E+09,9E+09]],
                                        [[0,0,0],[1,0,0,0],[0,-2,1,0],[0,9E+09,9E+09,9E+09,9E+09,9E+09]],
                                        [[0,0,0],[1,0,0,0],[0,-2,1,0],[0,9E+09,9E+09,9E+09,9E+09,9E+09]],
                                        [[0,0,0],[1,0,0,0],[0,-2,1,0],[0,9E+09,9E+09,9E+09,9E+09,9E+09]],
                                        [[0,0,0],[1,0,0,0],[0,-2,1,0],[0,9E+09,9E+09,9E+09,9E+09,9E+09]],
                                        [[0,0,0],[1,0,0,0],[0,-2,1,0],[0,9E+09,9E+09,9E+09,9E+09,9E+09]],
                                        [[0,0,0],[1,0,0,0],[0,-2,1,0],[0,9E+09,9E+09,9E+09,9E+09,9E+09]],
                                        [[0,0,0],[1,0,0,0],[0,-2,1,0],[0,9E+09,9E+09,9E+09,9E+09,9E+09]],
                                        [[0,0,0],[1,0,0,0],[0,-2,1,0],[0,9E+09,9E+09,9E+09,9E+09,9E+09]],
                                        [[0,0,0],[1,0,0,0],[0,-2,1,0],[0,9E+09,9E+09,9E+09,9E+09,9E+09]],
                                        [[0,0,0],[1,0,0,0],[0,-2,1,0],[0,9E+09,9E+09,9E+09,9E+09,9E+09]],
                                        [[0,0,0],[1,0,0,0],[0,-2,1,0],[0,9E+09,9E+09,9E+09,9E+09,9E+09]],
                                        [[0,0,0],[1,0,0,0],[0,-2,1,0],[0,9E+09,9E+09,9E+09,9E+09,9E+09]],
                                        [[0,0,0],[1,0,0,0],[0,-2,1,0],[0,9E+09,9E+09,9E+09,9E+09,9E+09]],
                                        [[0,0,0],[1,0,0,0],[0,-2,1,0],[0,9E+09,9E+09,9E+09,9E+09,9E+09]],
                                        [[0,0,0],[1,0,0,0],[0,-2,1,0],[0,9E+09,9E+09,9E+09,9E+09,9E+09]],
                                        [[0,0,0],[1,0,0,0],[0,-2,1,0],[0,9E+09,9E+09,9E+09,9E+09,9E+09]],
                                        [[0,0,0],[1,0,0,0],[0,-2,1,0],[0,9E+09,9E+09,9E+09,9E+09,9E+09]],
                                        [[0,0,0],[1,0,0,0],[0,-2,1,0],[0,9E+09,9E+09,9E+09,9E+09,9E+09]],
                                        [[0,0,0],[1,0,0,0],[0,-2,1,0],[0,9E+09,9E+09,9E+09,9E+09,9E+09]],
                                        [[0,0,0],[1,0,0,0],[0,-2,1,0],[0,9E+09,9E+09,9E+09,9E+09,9E+09]],
                                        [[0,0,0],[1,0,0,0],[0,-2,1,0],[0,9E+09,9E+09,9E+09,9E+09,9E+09]],
                                        [[0,0,0],[1,0,0,0],[0,-2,1,0],[0,9E+09,9E+09,9E+09,9E+09,9E+09]],
                                        [[0,0,0],[1,0,0,0],[0,-2,1,0],[0,9E+09,9E+09,9E+09,9E+09,9E+09]],
                                        [[0,0,0],[1,0,0,0],[0,-2,1,0],[0,9E+09,9E+09,9E+09,9E+09,9E+09]],
                                        [[0,0,0],[1,0,0,0],[0,-2,1,0],[0,9E+09,9E+09,9E+09,9E+09,9E+09]],
                                        [[0,0,0],[1,0,0,0],[0,-2,1,0],[0,9E+09,9E+09,9E+09,9E+09,9E+09]],
                                        [[0,0,0],[1,0,0,0],[0,-2,1,0],[0,9E+09,9E+09,9E+09,9E+09,9E+09]],
                                        [[0,0,0],[1,0,0,0],[0,-2,1,0],[0,9E+09,9E+09,9E+09,9E+09,9E+09]],
                                        [[0,0,0],[1,0,0,0],[0,-2,1,0],[0,9E+09,9E+09,9E+09,9E+09,9E+09]],
                                        [[0,0,0],[1,0,0,0],[0,-2,1,0],[0,9E+09,9E+09,9E+09,9E+09,9E+09]],
                                        [[0,0,0],[1,0,0,0],[0,-2,1,0],[0,9E+09,9E+09,9E+09,9E+09,9E+09]],
                                        [[0,0,0],[1,0,0,0],[0,-2,1,0],[0,9E+09,9E+09,9E+09,9E+09,9E+09]],
                                        [[0,0,0],[1,0,0,0],[0,-2,1,0],[0,9E+09,9E+09,9E+09,9E+09,9E+09]],
                                        [[0,0,0],[1,0,0,0],[0,-2,1,0],[0,9E+09,9E+09,9E+09,9E+09,9E+09]],
                                        [[0,0,0],[1,0,0,0],[0,-2,1,0],[0,9E+09,9E+09,9E+09,9E+09,9E+09]],
                                        [[0,0,0],[1,0,0,0],[0,-2,1,0],[0,9E+09,9E+09,9E+09,9E+09,9E+09]],
                                        [[0,0,0],[1,0,0,0],[0,-2,1,0],[0,9E+09,9E+09,9E+09,9E+09,9E+09]],
                                        [[0,0,0],[1,0,0,0],[0,-2,1,0],[0,9E+09,9E+09,9E+09,9E+09,9E+09]],
                                        [[0,0,0],[1,0,0,0],[0,-2,1,0],[0,9E+09,9E+09,9E+09,9E+09,9E+09]],
                                        [[0,0,0],[1,0,0,0],[0,-2,1,0],[0,9E+09,9E+09,9E+09,9E+09,9E+09]],
                                        [[0,0,0],[1,0,0,0],[0,-2,1,0],[0,9E+09,9E+09,9E+09,9E+09,9E+09]],
                                        [[0,0,0],[1,0,0,0],[0,-2,1,0],[0,9E+09,9E+09,9E+09,9E+09,9E+09]],
                                        [[0,0,0],[1,0,0,0],[0,-2,1,0],[0,9E+09,9E+09,9E+09,9E+09,9E+09]],
                                        [[0,0,0],[1,0,0,0],[0,-2,1,0],[0,9E+09,9E+09,9E+09,9E+09,9E+09]],
                                        [[0,0,0],[1,0,0,0],[0,-2,1,0],[0,9E+09,9E+09,9E+09,9E+09,9E+09]],
                                        [[0,0,0],[1,0,0,0],[0,-2,1,0],[0,9E+09,9E+09,9E+09,9E+09,9E+09]],
                                        [[0,0,0],[1,0,0,0],[0,-2,1,0],[0,9E+09,9E+09,9E+09,9E+09,9E+09]],
                                        [[0,0,0],[1,0,0,0],[0,-2,1,0],[0,9E+09,9E+09,9E+09,9E+09,9E+09]],
                                        [[0,0,0],[1,0,0,0],[0,-2,1,0],[0,9E+09,9E+09,9E+09,9E+09,9E+09]],
                                        [[0,0,0],[1,0,0,0],[0,-2,1,0],[0,9E+09,9E+09,9E+09,9E+09,9E+09]],
                                        [[0,0,0],[1,0,0,0],[0,-2,1,0],[0,9E+09,9E+09,9E+09,9E+09,9E+09]],
                                        [[0,0,0],[1,0,0,0],[0,-2,1,0],[0,9E+09,9E+09,9E+09,9E+09,9E+09]],
                                        [[0,0,0],[1,0,0,0],[0,-2,1,0],[0,9E+09,9E+09,9E+09,9E+09,9E+09]],
                                        [[0,0,0],[1,0,0,0],[0,-2,1,0],[0,9E+09,9E+09,9E+09,9E+09,9E+09]],
                                        [[0,0,0],[1,0,0,0],[0,-2,1,0],[0,9E+09,9E+09,9E+09,9E+09,9E+09]],
                                        [[0,0,0],[1,0,0,0],[0,-2,1,0],[0,9E+09,9E+09,9E+09,9E+09,9E+09]],
                                        [[0,0,0],[1,0,0,0],[0,-2,1,0],[0,9E+09,9E+09,9E+09,9E+09,9E+09]],
                                        [[0,0,0],[1,0,0,0],[0,-2,1,0],[0,9E+09,9E+09,9E+09,9E+09,9E+09]],
                                        [[0,0,0],[1,0,0,0],[0,-2,1,0],[0,9E+09,9E+09,9E+09,9E+09,9E+09]],
                                        [[0,0,0],[1,0,0,0],[0,-2,1,0],[0,9E+09,9E+09,9E+09,9E+09,9E+09]],
                                        [[0,0,0],[1,0,0,0],[0,-2,1,0],[0,9E+09,9E+09,9E+09,9E+09,9E+09]],
                                        [[0,0,0],[1,0,0,0],[0,-2,1,0],[0,9E+09,9E+09,9E+09,9E+09,9E+09]],
                                        [[0,0,0],[1,0,0,0],[0,-2,1,0],[0,9E+09,9E+09,9E+09,9E+09,9E+09]],
                                        [[0,0,0],[1,0,0,0],[0,-2,1,0],[0,9E+09,9E+09,9E+09,9E+09,9E+09]],
                                        [[0,0,0],[1,0,0,0],[0,-2,1,0],[0,9E+09,9E+09,9E+09,9E+09,9E+09]],
                                        [[0,0,0],[1,0,0,0],[0,-2,1,0],[0,9E+09,9E+09,9E+09,9E+09,9E+09]],
                                        [[0,0,0],[1,0,0,0],[0,-2,1,0],[0,9E+09,9E+09,9E+09,9E+09,9E+09]],
                                        [[0,0,0],[1,0,0,0],[0,-2,1,0],[0,9E+09,9E+09,9E+09,9E+09,9E+09]],
                                        [[0,0,0],[1,0,0,0],[0,-2,1,0],[0,9E+09,9E+09,9E+09,9E+09,9E+09]],
                                        [[0,0,0],[1,0,0,0],[0,-2,1,0],[0,9E+09,9E+09,9E+09,9E+09,9E+09]],
                                        [[0,0,0],[1,0,0,0],[0,-2,1,0],[0,9E+09,9E+09,9E+09,9E+09,9E+09]],
                                        [[0,0,0],[1,0,0,0],[0,-2,1,0],[0,9E+09,9E+09,9E+09,9E+09,9E+09]],
                                        [[0,0,0],[1,0,0,0],[0,-2,1,0],[0,9E+09,9E+09,9E+09,9E+09,9E+09]],
                                        [[0,0,0],[1,0,0,0],[0,-2,1,0],[0,9E+09,9E+09,9E+09,9E+09,9E+09]],
                                        [[0,0,0],[1,0,0,0],[0,-2,1,0],[0,9E+09,9E+09,9E+09,9E+09,9E+09]],
                                        [[0,0,0],[1,0,0,0],[0,-2,1,0],[0,9E+09,9E+09,9E+09,9E+09,9E+09]],
                                        [[0,0,0],[1,0,0,0],[0,-2,1,0],[0,9E+09,9E+09,9E+09,9E+09,9E+09]],
                                        [[0,0,0],[1,0,0,0],[0,-2,1,0],[0,9E+09,9E+09,9E+09,9E+09,9E+09]],
                                        [[0,0,0],[1,0,0,0],[0,-2,1,0],[0,9E+09,9E+09,9E+09,9E+09,9E+09]],
                                        [[0,0,0],[1,0,0,0],[0,-2,1,0],[0,9E+09,9E+09,9E+09,9E+09,9E+09]],
                                        [[0,0,0],[1,0,0,0],[0,-2,1,0],[0,9E+09,9E+09,9E+09,9E+09,9E+09]],
                                        [[0,0,0],[1,0,0,0],[0,-2,1,0],[0,9E+09,9E+09,9E+09,9E+09,9E+09]],
                                        [[0,0,0],[1,0,0,0],[0,-2,1,0],[0,9E+09,9E+09,9E+09,9E+09,9E+09]],
                                        [[0,0,0],[1,0,0,0],[0,-2,1,0],[0,9E+09,9E+09,9E+09,9E+09,9E+09]],
                                        [[0,0,0],[1,0,0,0],[0,-2,1,0],[0,9E+09,9E+09,9E+09,9E+09,9E+09]],
                                        [[0,0,0],[1,0,0,0],[0,-2,1,0],[0,9E+09,9E+09,9E+09,9E+09,9E+09]],
                                        [[0,0,0],[1,0,0,0],[0,-2,1,0],[0,9E+09,9E+09,9E+09,9E+09,9E+09]],
                                        [[0,0,0],[1,0,0,0],[0,-2,1,0],[0,9E+09,9E+09,9E+09,9E+09,9E+09]],
                                        [[0,0,0],[1,0,0,0],[0,-2,1,0],[0,9E+09,9E+09,9E+09,9E+09,9E+09]],
                                        [[0,0,0],[1,0,0,0],[0,-2,1,0],[0,9E+09,9E+09,9E+09,9E+09,9E+09]],
                                        [[0,0,0],[1,0,0,0],[0,-2,1,0],[0,9E+09,9E+09,9E+09,9E+09,9E+09]],
                                        [[0,0,0],[1,0,0,0],[0,-2,1,0],[0,9E+09,9E+09,9E+09,9E+09,9E+09]],
                                        [[0,0,0],[1,0,0,0],[0,-2,1,0],[0,9E+09,9E+09,9E+09,9E+09,9E+09]],
                                        [[0,0,0],[1,0,0,0],[0,-2,1,0],[0,9E+09,9E+09,9E+09,9E+09,9E+09]],
                                        [[0,0,0],[1,0,0,0],[0,-2,1,0],[0,9E+09,9E+09,9E+09,9E+09,9E+09]],
                                        [[0,0,0],[1,0,0,0],[0,-2,1,0],[0,9E+09,9E+09,9E+09,9E+09,9E+09]],
                                        [[0,0,0],[1,0,0,0],[0,-2,1,0],[0,9E+09,9E+09,9E+09,9E+09,9E+09]],
                                        [[0,0,0],[1,0,0,0],[0,-2,1,0],[0,9E+09,9E+09,9E+09,9E+09,9E+09]],
                                        [[0,0,0],[1,0,0,0],[0,-2,1,0],[0,9E+09,9E+09,9E+09,9E+09,9E+09]],
                                        [[0,0,0],[1,0,0,0],[0,-2,1,0],[0,9E+09,9E+09,9E+09,9E+09,9E+09]],
                                        [[0,0,0],[1,0,0,0],[0,-2,1,0],[0,9E+09,9E+09,9E+09,9E+09,9E+09]],
                                        [[0,0,0],[1,0,0,0],[0,-2,1,0],[0,9E+09,9E+09,9E+09,9E+09,9E+09]],
                                        [[0,0,0],[1,0,0,0],[0,-2,1,0],[0,9E+09,9E+09,9E+09,9E+09,9E+09]],
                                        [[0,0,0],[1,0,0,0],[0,-2,1,0],[0,9E+09,9E+09,9E+09,9E+09,9E+09]],
                                        [[0,0,0],[1,0,0,0],[0,-2,1,0],[0,9E+09,9E+09,9E+09,9E+09,9E+09]],
                                        [[0,0,0],[1,0,0,0],[0,-2,1,0],[0,9E+09,9E+09,9E+09,9E+09,9E+09]],
                                        [[0,0,0],[1,0,0,0],[0,-2,1,0],[0,9E+09,9E+09,9E+09,9E+09,9E+09]],
                                        [[0,0,0],[1,0,0,0],[0,-2,1,0],[0,9E+09,9E+09,9E+09,9E+09,9E+09]],
                                        [[0,0,0],[1,0,0,0],[0,-2,1,0],[0,9E+09,9E+09,9E+09,9E+09,9E+09]],
                                        [[0,0,0],[1,0,0,0],[0,-2,1,0],[0,9E+09,9E+09,9E+09,9E+09,9E+09]],
                                        [[0,0,0],[1,0,0,0],[0,-2,1,0],[0,9E+09,9E+09,9E+09,9E+09,9E+09]],
                                        [[0,0,0],[1,0,0,0],[0,-2,1,0],[0,9E+09,9E+09,9E+09,9E+09,9E+09]],
                                        [[0,0,0],[1,0,0,0],[0,-2,1,0],[0,9E+09,9E+09,9E+09,9E+09,9E+09]],
                                        [[0,0,0],[1,0,0,0],[0,-2,1,0],[0,9E+09,9E+09,9E+09,9E+09,9E+09]],
                                        [[0,0,0],[1,0,0,0],[0,-2,1,0],[0,9E+09,9E+09,9E+09,9E+09,9E+09]],
                                        [[0,0,0],[1,0,0,0],[0,-2,1,0],[0,9E+09,9E+09,9E+09,9E+09,9E+09]],
                                        [[0,0,0],[1,0,0,0],[0,-2,1,0],[0,9E+09,9E+09,9E+09,9E+09,9E+09]],
                                        [[0,0,0],[1,0,0,0],[0,-2,1,0],[0,9E+09,9E+09,9E+09,9E+09,9E+09]],
                                        [[0,0,0],[1,0,0,0],[0,-2,1,0],[0,9E+09,9E+09,9E+09,9E+09,9E+09]],
                                        [[0,0,0],[1,0,0,0],[0,-2,1,0],[0,9E+09,9E+09,9E+09,9E+09,9E+09]],
                                        [[0,0,0],[1,0,0,0],[0,-2,1,0],[0,9E+09,9E+09,9E+09,9E+09,9E+09]],
                                        [[0,0,0],[1,0,0,0],[0,-2,1,0],[0,9E+09,9E+09,9E+09,9E+09,9E+09]],
                                        [[0,0,0],[1,0,0,0],[0,-2,1,0],[0,9E+09,9E+09,9E+09,9E+09,9E+09]],
                                        [[0,0,0],[1,0,0,0],[0,-2,1,0],[0,9E+09,9E+09,9E+09,9E+09,9E+09]],
                                        [[0,0,0],[1,0,0,0],[0,-2,1,0],[0,9E+09,9E+09,9E+09,9E+09,9E+09]],
                                        [[0,0,0],[1,0,0,0],[0,-2,1,0],[0,9E+09,9E+09,9E+09,9E+09,9E+09]],
                                        [[0,0,0],[1,0,0,0],[0,-2,1,0],[0,9E+09,9E+09,9E+09,9E+09,9E+09]],
                                        [[0,0,0],[1,0,0,0],[0,-2,1,0],[0,9E+09,9E+09,9E+09,9E+09,9E+09]],
                                        [[0,0,0],[1,0,0,0],[0,-2,1,0],[0,9E+09,9E+09,9E+09,9E+09,9E+09]],
                                        [[0,0,0],[1,0,0,0],[0,-2,1,0],[0,9E+09,9E+09,9E+09,9E+09,9E+09]],
                                        [[0,0,0],[1,0,0,0],[0,-2,1,0],[0,9E+09,9E+09,9E+09,9E+09,9E+09]],
                                        [[0,0,0],[1,0,0,0],[0,-2,1,0],[0,9E+09,9E+09,9E+09,9E+09,9E+09]],
                                        [[0,0,0],[1,0,0,0],[0,-2,1,0],[0,9E+09,9E+09,9E+09,9E+09,9E+09]],
                                        [[0,0,0],[1,0,0,0],[0,-2,1,0],[0,9E+09,9E+09,9E+09,9E+09,9E+09]],
                                        [[0,0,0],[1,0,0,0],[0,-2,1,0],[0,9E+09,9E+09,9E+09,9E+09,9E+09]],
                                        [[0,0,0],[1,0,0,0],[0,-2,1,0],[0,9E+09,9E+09,9E+09,9E+09,9E+09]],
                                        [[0,0,0],[1,0,0,0],[0,-2,1,0],[0,9E+09,9E+09,9E+09,9E+09,9E+09]],
                                        [[0,0,0],[1,0,0,0],[0,-2,1,0],[0,9E+09,9E+09,9E+09,9E+09,9E+09]],
                                        [[0,0,0],[1,0,0,0],[0,-2,1,0],[0,9E+09,9E+09,9E+09,9E+09,9E+09]],
                                        [[0,0,0],[1,0,0,0],[0,-2,1,0],[0,9E+09,9E+09,9E+09,9E+09,9E+09]],
                                        [[0,0,0],[1,0,0,0],[0,-2,1,0],[0,9E+09,9E+09,9E+09,9E+09,9E+09]],
                                        [[0,0,0],[1,0,0,0],[0,-2,1,0],[0,9E+09,9E+09,9E+09,9E+09,9E+09]],
                                        [[0,0,0],[1,0,0,0],[0,-2,1,0],[0,9E+09,9E+09,9E+09,9E+09,9E+09]],
                                        [[0,0,0],[1,0,0,0],[0,-2,1,0],[0,9E+09,9E+09,9E+09,9E+09,9E+09]],
                                        [[0,0,0],[1,0,0,0],[0,-2,1,0],[0,9E+09,9E+09,9E+09,9E+09,9E+09]],
                                        [[0,0,0],[1,0,0,0],[0,-2,1,0],[0,9E+09,9E+09,9E+09,9E+09,9E+09]],
                                        [[0,0,0],[1,0,0,0],[0,-2,1,0],[0,9E+09,9E+09,9E+09,9E+09,9E+09]],
                                        [[0,0,0],[1,0,0,0],[0,-2,1,0],[0,9E+09,9E+09,9E+09,9E+09,9E+09]],
                                        [[0,0,0],[1,0,0,0],[0,-2,1,0],[0,9E+09,9E+09,9E+09,9E+09,9E+09]],
                                        [[0,0,0],[1,0,0,0],[0,-2,1,0],[0,9E+09,9E+09,9E+09,9E+09,9E+09]],
                                        [[0,0,0],[1,0,0,0],[0,-2,1,0],[0,9E+09,9E+09,9E+09,9E+09,9E+09]],
                                        [[0,0,0],[1,0,0,0],[0,-2,1,0],[0,9E+09,9E+09,9E+09,9E+09,9E+09]],
                                        [[0,0,0],[1,0,0,0],[0,-2,1,0],[0,9E+09,9E+09,9E+09,9E+09,9E+09]],
                                        [[0,0,0],[1,0,0,0],[0,-2,1,0],[0,9E+09,9E+09,9E+09,9E+09,9E+09]],
                                        [[100,200,300],[1,0,0,0],[0,0,0,0],[9E+09,9E+09,9E+09,9E+09,9E+09,9E+09]],
                                        [[100,200,300],[1,0,0,0],[0,0,0,0],[9E+09,9E+09,9E+09,9E+09,9E+09,9E+09]],
                                        [[100,200,300],[1,0,0,0],[0,0,0,0],[9E+09,9E+09,9E+09,9E+09,9E+09,9E+09]],
                                        [[100,200,300],[1,0,0,0],[0,0,0,0],[9E+09,9E+09,9E+09,9E+09,9E+09,9E+09]],
                                        [[100,200,300],[1,0,0,0],[0,0,0,0],[9E+09,9E+09,9E+09,9E+09,9E+09,9E+09]],
                                        [[100,200,300],[1,0,0,0],[0,0,0,0],[9E+09,9E+09,9E+09,9E+09,9E+09,9E+09]],
                                        [[100,200,300],[1,0,0,0],[0,0,0,0],[9E+09,9E+09,9E+09,9E+09,9E+09,9E+09]],
                                        [[100,200,300],[1,0,0,0],[0,0,0,0],[9E+09,9E+09,9E+09,9E+09,9E+09,9E+09]],
                                        [[100,200,300],[1,0,0,0],[0,0,0,0],[9E+09,9E+09,9E+09,9E+09,9E+09,9E+09]],
                                        [[100,200,300],[1,0,0,0],[0,0,0,0],[9E+09,9E+09,9E+09,9E+09,9E+09,9E+09]],
                                        [[100,200,300],[1,0,0,0],[0,0,0,0],[9E+09,9E+09,9E+09,9E+09,9E+09,9E+09]],
                                        [[100,200,300],[1,0,0,0],[0,0,0,0],[9E+09,9E+09,9E+09,9E+09,9E+09,9E+09]],
                                        [[100,200,300],[1,0,0,0],[0,0,0,0],[9E+09,9E+09,9E+09,9E+09,9E+09,9E+09]],
                                        [[100,200,300],[1,0,0,0],[0,0,0,0],[9E+09,9E+09,9E+09,9E+09,9E+09,9E+09]],
                                        [[100,200,300],[1,0,0,0],[0,0,0,0],[9E+09,9E+09,9E+09,9E+09,9E+09,9E+09]],
                                        [[100,200,300],[1,0,0,0],[0,0,0,0],[9E+09,9E+09,9E+09,9E+09,9E+09,9E+09]],
                                        [[100,200,300],[1,0,0,0],[0,0,0,0],[9E+09,9E+09,9E+09,9E+09,9E+09,9E+09]],
                                        [[100,200,300],[1,0,0,0],[0,0,0,0],[9E+09,9E+09,9E+09,9E+09,9E+09,9E+09]],
                                        [[100,200,300],[1,0,0,0],[0,0,0,0],[9E+09,9E+09,9E+09,9E+09,9E+09,9E+09]],
                                        [[100,200,300],[1,0,0,0],[0,0,0,0],[9E+09,9E+09,9E+09,9E+09,9E+09,9E+09]],
                                        [[100,200,300],[1,0,0,0],[0,0,0,0],[9E+09,9E+09,9E+09,9E+09,9E+09,9E+09]],
                                        [[100,200,300],[1,0,0,0],[0,0,0,0],[9E+09,9E+09,9E+09,9E+09,9E+09,9E+09]],
                                        [[100,200,300],[1,0,0,0],[0,0,0,0],[9E+09,9E+09,9E+09,9E+09,9E+09,9E+09]],
                                        [[100,200,300],[1,0,0,0],[0,0,0,0],[9E+09,9E+09,9E+09,9E+09,9E+09,9E+09]],
                                        [[100,200,300],[1,0,0,0],[0,0,0,0],[9E+09,9E+09,9E+09,9E+09,9E+09,9E+09]],
                                        [[100,200,300],[1,0,0,0],[0,0,0,0],[9E+09,9E+09,9E+09,9E+09,9E+09,9E+09]],
                                        [[100,200,300],[1,0,0,0],[0,0,0,0],[9E+09,9E+09,9E+09,9E+09,9E+09,9E+09]],
                                        [[100,200,300],[1,0,0,0],[0,0,0,0],[9E+09,9E+09,9E+09,9E+09,9E+09,9E+09]],
                                        [[100,200,300],[1,0,0,0],[0,0,0,0],[9E+09,9E+09,9E+09,9E+09,9E+09,9E+09]],
                                        [[100,200,300],[1,0,0,0],[0,0,0,0],[9E+09,9E+09,9E+09,9E+09,9E+09,9E+09]],
                                        [[100,200,300],[1,0,0,0],[0,0,0,0],[9E+09,9E+09,9E+09,9E+09,9E+09,9E+09]],
                                        [[100,200,300],[1,0,0,0],[0,0,0,0],[9E+09,9E+09,9E+09,9E+09,9E+09,9E+09]],
                                        [[100,200,300],[1,0,0,0],[0,0,0,0],[9E+09,9E+09,9E+09,9E+09,9E+09,9E+09]],
                                        [[100,200,300],[1,0,0,0],[0,0,0,0],[9E+09,9E+09,9E+09,9E+09,9E+09,9E+09]],
                                        [[100,200,300],[1,0,0,0],[0,0,0,0],[9E+09,9E+09,9E+09,9E+09,9E+09,9E+09]],
                                        [[100,200,300],[1,0,0,0],[0,0,0,0],[9E+09,9E+09,9E+09,9E+09,9E+09,9E+09]],
                                        [[100,200,300],[1,0,0,0],[0,0,0,0],[9E+09,9E+09,9E+09,9E+09,9E+09,9E+09]],
                                        [[100,200,300],[1,0,0,0],[0,0,0,0],[9E+09,9E+09,9E+09,9E+09,9E+09,9E+09]],
                                        [[100,200,300],[1,0,0,0],[0,0,0,0],[9E+09,9E+09,9E+09,9E+09,9E+09,9E+09]],
                                        [[100,200,300],[1,0,0,0],[0,0,0,0],[9E+09,9E+09,9E+09,9E+09,9E+09,9E+09]],
                                        [[100,200,300],[1,0,0,0],[0,0,0,0],[9E+09,9E+09,9E+09,9E+09,9E+09,9E+09]],
                                        [[100,200,300],[1,0,0,0],[0,0,0,0],[9E+09,9E+09,9E+09,9E+09,9E+09,9E+09]],
                                        [[100,200,300],[1,0,0,0],[0,0,0,0],[9E+09,9E+09,9E+09,9E+09,9E+09,9E+09]],
                                        [[100,200,300],[1,0,0,0],[0,0,0,0],[9E+09,9E+09,9E+09,9E+09,9E+09,9E+09]],
                                        [[100,200,300],[1,0,0,0],[0,0,0,0],[9E+09,9E+09,9E+09,9E+09,9E+09,9E+09]],
                                        [[100,200,300],[1,0,0,0],[0,0,0,0],[9E+09,9E+09,9E+09,9E+09,9E+09,9E+09]],
                                        [[100,200,300],[1,0,0,0],[0,0,0,0],[9E+09,9E+09,9E+09,9E+09,9E+09,9E+09]],
                                        [[100,200,300],[1,0,0,0],[0,0,0,0],[9E+09,9E+09,9E+09,9E+09,9E+09,9E+09]],
                                        [[100,200,300],[1,0,0,0],[0,0,0,0],[9E+09,9E+09,9E+09,9E+09,9E+09,9E+09]],
                                        [[100,200,300],[1,0,0,0],[0,0,0,0],[9E+09,9E+09,9E+09,9E+09,9E+09,9E+09]],
                                        [[100,200,300],[1,0,0,0],[0,0,0,0],[9E+09,9E+09,9E+09,9E+09,9E+09,9E+09]],
                                        [[100,200,300],[1,0,0,0],[0,0,0,0],[9E+09,9E+09,9E+09,9E+09,9E+09,9E+09]],
                                        [[100,200,300],[1,0,0,0],[0,0,0,0],[9E+09,9E+09,9E+09,9E+09,9E+09,9E+09]],
                                        [[100,200,300],[1,0,0,0],[0,0,0,0],[9E+09,9E+09,9E+09,9E+09,9E+09,9E+09]],
                                        [[100,200,300],[1,0,0,0],[0,0,0,0],[9E+09,9E+09,9E+09,9E+09,9E+09,9E+09]],
                                        [[100,200,300],[1,0,0,0],[0,0,0,0],[9E+09,9E+09,9E+09,9E+09,9E+09,9E+09]],
                                        [[100,200,300],[1,0,0,0],[0,0,0,0],[9E+09,9E+09,9E+09,9E+09,9E+09,9E+09]],
                                        [[100,200,300],[1,0,0,0],[0,0,0,0],[9E+09,9E+09,9E+09,9E+09,9E+09,9E+09]],
                                        [[100,200,300],[1,0,0,0],[0,0,0,0],[9E+09,9E+09,9E+09,9E+09,9E+09,9E+09]],
                                        [[100,200,300],[1,0,0,0],[0,0,0,0],[9E+09,9E+09,9E+09,9E+09,9E+09,9E+09]],
                                        [[100,200,300],[1,0,0,0],[0,0,0,0],[9E+09,9E+09,9E+09,9E+09,9E+09,9E+09]],
                                        [[100,200,300],[1,0,0,0],[0,0,0,0],[9E+09,9E+09,9E+09,9E+09,9E+09,9E+09]],
                                        [[100,200,300],[1,0,0,0],[0,0,0,0],[9E+09,9E+09,9E+09,9E+09,9E+09,9E+09]],
                                        [[100,200,300],[1,0,0,0],[0,0,0,0],[9E+09,9E+09,9E+09,9E+09,9E+09,9E+09]],
                                        [[100,200,300],[1,0,0,0],[0,0,0,0],[9E+09,9E+09,9E+09,9E+09,9E+09,9E+09]],
